(*AlarmCtrl*)
(*============================*)
//AlarmCtrl();
Alarm_IO();
Alarm_Others();
MisshookSensorCtrl();
(*Arm2MisshookSensorCtrl();*)
DeactivateCtrl();

(*AnalogCtrl*)
(*============================*)
(*BrensonGen_AnalogDigitalCtrl();*)
(*BrensonMultiFreq_Main();*)
(*USFeedbackCtrl();*)
ClangsonicUSCommCtrl();
ClangsonicUSCtrl();
ModbusControl_ST();
MegasonicModbusProgram_ST();
ClangsonicUSModbusFeedbackCtrl();
ConductivityCtrl();
FilterPressureCtrl();
TempChillerCtrl();
TempCtrl();
PID_TempCtrl();
//PIDCtrl();

(*AutoArmCtrl*)
(*============================*)
VertCoERead();
HorzCoeRead();
SlowpullCoeRead();
OmronServoEnable();
AxisHorzAdditionalInterlock_Arm1();
AxisServoCtrl_SlowPull();
oArmSlowPullHomingCtrl();
oArmSlowPullOutputCtrl();
PosConfirmBitCtrl_SlowPull();

AxisHorzMovementOutputCtrl_Arm1();
AxisServoCtrl_Arm1();
AxisServoCtrlMapping_Arm1();
AxisVertMovementOutputCtrl_Arm1();
PnpCtrl_Arm1();
PnpMapping_Arm1();
PnPstorageMemory_Arm();
PosConfirmBitCtrl_Arm1();

(*PosConfirmBitCtrl_SlowPull();*)
(*AxisHorzAdditionalInterlock_Arm1();*)
(*AxisHorzOutputCtrlInterlockingST_Arm1();*)
(*AxisMovementOutputCtrl_SlowPull();*)
(*AxisServoCtrl_SlowPull();*)
(*AutoProcessCtrl*)

(*============================*)
LdBasketMissingCtrl();
LdPrcs();
LdPrcs_General();
Stn1();
Stn2();
Stn3();
Stn4();
Stn5();
Stn6();
Stn7();
Stn7ReturnPumpCtrl();
Stn8();
Stn9();
Stn9SlowPullCalculation();
Stn10();
//Lift_N_Shuttle();
BarcodeCtrl_Utac();
BarcodeScanner();
Cascading();
StnOverflowValveCtrl();

(*AutoSevenDayOnOffCtrl*)
(*============================*)
SevenDayCtrl();
SevenDayOnOffConf();

(*BaseWork*)
(*============================*)
TowerLightCtrl();
UserCtrl();

(*BasketMemory_RecipeCtrl*)
(*============================*)
BasketBadCtrl();
BasketMemoryCtrl();
BasketToleranceCtrl();
BskMemoryCtrl();
CvMotorREFE();

(*BlowerCtrl*)
(*============================*)
//BlowerCtrl();

(*DataManagement*)
(*============================*)
ArmPickTransferCtrl_General();
BasketTotalizer();
MacOperationTimeCtrl();
RTClockCtrl();
StnBasketTotalizer();

(* CSV *)
Batch_Number_counter();
Csv_Report_Ctrl();
Csv_Report_Mapping();

(*DataManagement_Barcode*)
(*============================*)
//Batch_Number_counter();
//GeneratorComparison();
Log_BasketTimeInOut();
Log_Configuration();
Log_Management();

(*DosingPumpCtrl*)
(*============================*)
ManualDosingSTreset();
Stn1DosingPumpCtrl();
(*Stn2DosingPumpCtrl();*)
Stn3DosingPumpCtrl();
(*Stn4DosingPumpCtrl();*)
Stn5DosingPumpCtrl();

(*ManualCtrl*)
(*============================*)
ManualButtonCtrl();
ManualCtrl();
ManualCtrl_Arm();
ManualLifterJog();

(*Other*)
(*============================*)
ArmXYPosAdjust();
BeckhoffHMIMapping();
HMI_Function();
HoldingBit_DoorTransfer();
HoldingBitCtrl();
(*IndusoftBeckhoffMapping();*)
ProHMIMapping();
TactTime();
zHMIMaxMinLimit();
ClockPulse10ms();

(*OutputCtrl*)
(*============================*)
MAIN_Arm_Mapping();
MP_1_Y100();
MP_2_Y101();
MP_3_Y102();
MP_4_Y103();
SP1_1_Y110();
SP1_2_Y111();
SP2_1_Y120();
SP3_1_Y130();
SP3_2_Y131();
SP3_3_Y132();
STN_TopUpCtrl();


(*TimeOptimize*)
(*============================*)
Optimizer_Monitor();
TimeOptimizeCtrl();
TimeTrackerCtrl();

(*HMI*)
HMI_Ctrl();
StartStop();

HMI_CKK();


(*xml_Function*)
(*============================*)
//Xml_AddressMapping();
//XML_Program();
pouXMLRecipeTest();




	tPowerOnDelayOn(IN:=TRUE , PT:=T#5S , Q=> , ET=> );
	tPowerOnDelayOff(IN:=tPowerOnDelayOn.Q , PT:=t#2s , Q=> , ET=> );
	
	IF bRecipeLoadPB OR (tPowerOnDelayOn.Q AND NOT tPowerOnDelayOff.Q) THEN
	bRecipeLoadInternal := TRUE;
	bRecipeLoadPB := FALSE;
	ELSE
	bRecipeLoadInternal := FALSE;
	END_IF

//END_IF

END_PROGRAM

// ---- POUs/MainProgram/XML/Bootup_Shutdown_ctrl.TcPOU
PROGRAM Bootup_Shutdown_ctrl
VAR
	bIpcInput_on: BOOL;
	bXmlReadEn: BOOL;
	bCSVReadEn: BOOL;
	bCsvReadDone: BOOL;
	
	bIPCInputOnRE	: R_trig;
	bIPCOnRE		: R_Trig;
	bXmlCsvReadDoneRE : R_Trig;
	bXmlCsvWriteDoneRE	:R_trig;
	
	bCsvWriteEn: BOOL;
	bIpcOnHR: BOOL;


	
	bSFQTest: BOOL;
	bSFQTest_read: BOOL;
	

	bBootUpReadXMLDone	:BOOL;
	bShutdownWriteXMLDone	:BOOL;
	sStatus: STRING;
	bsyed: BOOL;
	bIpcOffDelay: BOOL;
	tIpcOffDelay: TON;
	test: Bool;
	
	
	
	
	
	
	
	

	
	
	
	
	bSHutdownTest: BOOL;
	
	on: BOOL;


END_VAR

VAR PERSISTENT
	bBootupHold: BOOL;
END_VAR


// IPC OFF Selector Switch - OFF
bIPCInputOnRE(CLK:=ARbDI[eX11111_IpcDcOnSignal] OR bBatteryModeActivated OR bSFQTest , Q=> );

IF ARbDI[eX11111_IpcDcOnSignal] THEN
	on:= FALSE;
	ELSE
	on:= TRUE;
	
END_IF


// IPC autoboot start signal
bIPCOnRE(CLK:=TRUE OR bSFQTest_read  , Q=> );

//IPC On Holding relay -output
IF PowerOnDelay.Q AND NOT tIpcOffDelay.Q THEN
	bIpcOnHR := TRUE;
	ELSE
	bIpcOnHR := FALSE;
END_IF

ARwDO[eY11007_IpcDcOnHoldingRelay].00:=bIpcOnHR OR bsyed;

// Bootup
IF bIPCOnRE.Q AND NOT bBootupHold THEN
	bMainCtrl:=FALSE;
	bReadXmlEn:= TRUE;
END_IF

bXmlCsvReadDoneRE(CLK:= bReadXmlComplete (*AND NOT Alarm_XMLReadnWrite.fbXmlSrvReadFromXML.bBusy AND bCsvReadDone*) , Q=> );

IF bXmlCsvReadDoneRE.Q THEN 
	bMainCtrl:=TRUE;
	bBootupHold:= TRUE;
END_IF

// Shutdown
IF bIPCInputOnRE.Q OR bSHutdownTest THEN
	bBootupHold:= FALSE;
	bMachineShutdown:=TRUE;
	bShutdownPopupPage:=TRUE;
	bRecipeShutdownRequestFlag:= TRUE;
	bCsvShutdownRequestFlag:=TRUE;
	bWriteXmlEn:= TRUE;
END_IF

bXmlCsvWriteDoneRE(CLK:= bWrite_Done (*AND bRecipeReadyToShutdownFlag AND bCsvReadyToShutdownFlag*), Q=> );

IF bXmlCsvWriteDoneRE.Q THEN
	bIpcOffDelay:= TRUE;
	bWriteXmlEn:=FALSE;
	
END_IF

tIpcOffDelay(IN:=bIpcOffDelay , PT:= T#2S , Q=> , ET=> );

END_PROGRAM

// ---- POUs/MainProgram/Barcode/SerialCom.TcPOU
PROGRAM SerialCom
VAR
	fbSerialControl : SerialLineControlADS;
	fbSendString	: SendString;
	fbReceiveString	: ReceiveString;
	
	bBarcodeReceivedReset_FE: F_TRIG;
END_VAR

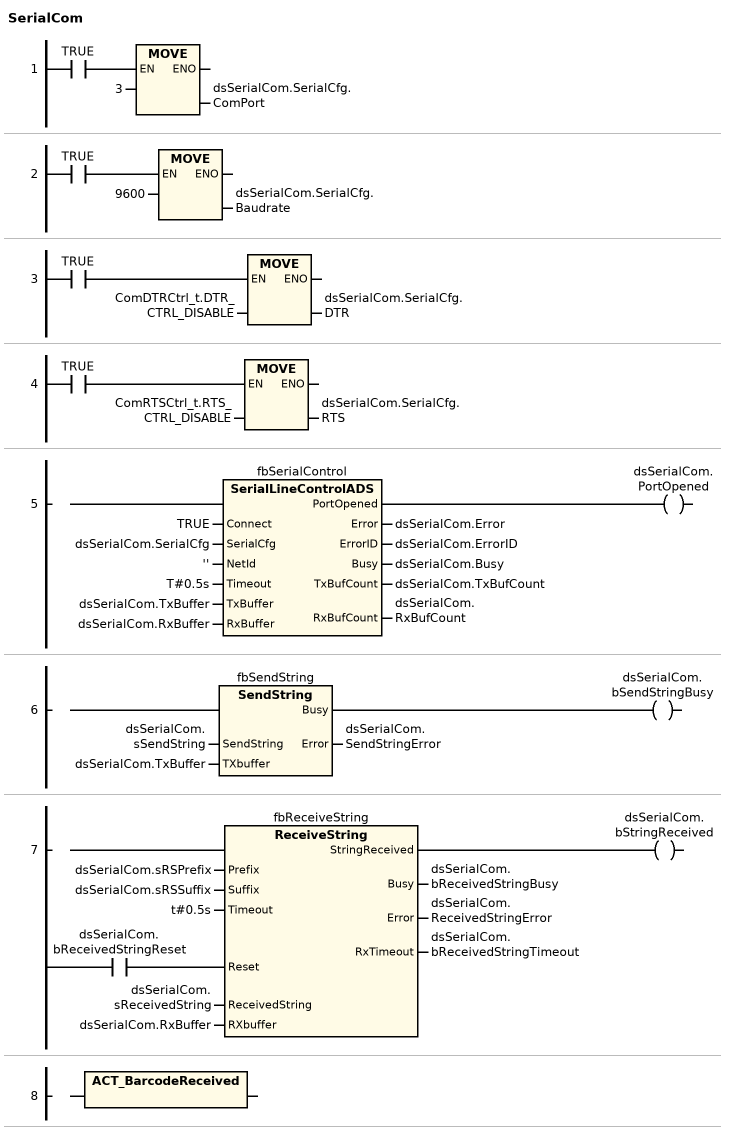
// NETWORK 1
dsSerialCom.SerialCfg.ComPort := 3;

// NETWORK 2
dsSerialCom.SerialCfg.Baudrate := 9600;

// NETWORK 3
dsSerialCom.SerialCfg.DTR := ComDTRCtrl_t.DTR_CTRL_DISABLE;

// NETWORK 4
dsSerialCom.SerialCfg.RTS := ComRTSCtrl_t.RTS_CTRL_DISABLE;

// NETWORK 5
fbSerialControl(
    Connect := TRUE,
    SerialCfg := dsSerialCom.SerialCfg,
    NetId := '',
    Timeout := T#0.5s,
    TxBuffer := dsSerialCom.TxBuffer,
    RxBuffer := dsSerialCom.RxBuffer,
    Error => dsSerialCom.Error,
    ErrorID => dsSerialCom.ErrorID,
    Busy => dsSerialCom.Busy,
    TxBufCount => dsSerialCom.TxBufCount,
    RxBufCount => dsSerialCom.RxBufCount); // SerialLineControlADS
dsSerialCom.PortOpened := fbSerialControl.PortOpened;

// NETWORK 6
fbSendString(
    SendString := dsSerialCom.sSendString,
    TXbuffer := dsSerialCom.TxBuffer,
    Error => dsSerialCom.SendStringError); // SendString
dsSerialCom.bSendStringBusy := fbSendString.Busy;

// NETWORK 7
fbReceiveString(
    Prefix := dsSerialCom.sRSPrefix,
    Suffix := dsSerialCom.sRSSuffix,
    Timeout := t#0.5s,
    Reset := dsSerialCom.bReceivedStringReset,
    ReceivedString := dsSerialCom.sReceivedString,
    RXbuffer := dsSerialCom.RxBuffer,
    Busy => dsSerialCom.bReceivedStringBusy,
    Error => dsSerialCom.ReceivedStringError,
    RxTimeout => dsSerialCom.bReceivedStringTimeout); // ReceiveString
dsSerialCom.bStringReceived := fbReceiveString.StringReceived;

// NETWORK 8
ACT_BarcodeReceived();

ACTION ACT_BarcodeReceived:

bBarcodeReceivedReset_FE(CLK:=((bAutoStartPb AND ARbDI[eX14000_LoadingConveyorSensor_Feed]) OR bBarcodeRegPage), Q=> );

IF bBarcodeReceivedReset_FE.Q THEN
dsSerialCom.sReceivedString:='';
END_IF
END_ACTION

END_PROGRAM

// ---- POUs/MainProgram/OPC_UA/OPC_UA_MAP.TcPOU
PROGRAM OPC_UA_MAP
VAR
	bIPC_Machine_Run: BOOL;
	bIPC_Machine_Alarm: BOOL;
	bIPC_Ideal_Cycle_Time: INT;


END_VAR

bMachine_Run_OPC_UA 	:=bAutoStartPb;			
                                    
                                    
bMachine_Idle_OPC_UA 	:=ARwDO[eY11005_GeneralTowerLightInd_Yellow].00;			
                                    
                                    
bMachine_Alarm_OPC_UA 	:=ARwDO[eY11004_GeneralTowerLightInd_Red].00;			
                                    
                                    
iRecipe_Number_OPC_UA 	:=iUserDefineProductRecipeNo;				
                                    
                                    
sUsername_OPCUA 		:=fbHmiTF1800_UserlevelManagement.dsHmiUserStatus_Active.sLoginName;				
                                    
                                    
ARbBasketAvailibility_OPCUA[1]:= DSStnBasketInfo[1].bAvailibility;			
ARbBasketAvailibility_OPCUA[2]:= DSStnBasketInfo[2].bAvailibility;;
ARbBasketAvailibility_OPCUA[3]:= DSStnBasketInfo[3].bAvailibility;;
ARbBasketAvailibility_OPCUA[4]:= DSStnBasketInfo[4].bAvailibility;;
ARbBasketAvailibility_OPCUA[5]:= DSStnBasketInfo[5].bAvailibility;;
ARbBasketAvailibility_OPCUA[6]:= DSStnBasketInfo[6].bAvailibility;;
ARbBasketAvailibility_OPCUA[7]:= DSStnBasketInfo[7].bAvailibility;;
ARbBasketAvailibility_OPCUA[8]:= DSStnBasketInfo[8].bAvailibility;;
ARbBasketAvailibility_OPCUA[9]:= DSStnBasketInfo[9].bAvailibility;;
//ARbBasketAvailibility_OPCUA[10]:= DSStnBasketInfo[10].bAvailibility;;
                                    
                                    
ARbStationBasketStatus_OPCUA[1]:=DSStnBasketInfo[1].sProductQuality;			
ARbStationBasketStatus_OPCUA[2]:=DSStnBasketInfo[2].sProductQuality;                                    
ARbStationBasketStatus_OPCUA[3]:=DSStnBasketInfo[3].sProductQuality;                                    
ARbStationBasketStatus_OPCUA[4]:=DSStnBasketInfo[4].sProductQuality;
ARbStationBasketStatus_OPCUA[5]:=DSStnBasketInfo[5].sProductQuality;
ARbStationBasketStatus_OPCUA[6]:=DSStnBasketInfo[6].sProductQuality;
ARbStationBasketStatus_OPCUA[7]:=DSStnBasketInfo[7].sProductQuality;
ARbStationBasketStatus_OPCUA[8]:=DSStnBasketInfo[8].sProductQuality;
ARbStationBasketStatus_OPCUA[9]:=DSStnBasketInfo[9].sProductQuality;
//ARbStationBasketStatus_OPCUA[10]:=DSStnBasketInfo[10].sProductQuality;

                                    
                                    
ARrStnTempPV_OPCUA					:=ARrStnTempPV;                                
                                  
ARrStnTempHysterysisSV_OPCUA		:=ARrStnTempHYSsv;			                                    	
                                    
ARrStnTempHighTempSV_OPCUA			:=ARrStnTempHALsv;			                                  	
                                    
ARrStnTempSV_OPCUA					:=ARrStnTempSV;					                                    
                                    
ARrStnTempReadySV_OPCUA				:=ARrStnTempRDYsv;		                                    
                                    
ARrStnTemp1stLimitSV_OPCUA			:=ARrStnTemp1stLimitSv;	
                                   
ARrStnTemp2ndLimitSV_OPCUA			:=ARrStnTemp2ndLimitSv;		                                    
                                 
ARiStnPreparationTempSV_OPCUA		:=ARiStnPreparationTempSv;
                                                                      
ARrStnConductivityPV_OPCUA 			:=ARrStnConductivityPV;
                                                                      
ARrStnLowConductivitySV_OPCUA		:=ARrStnLowConductivitySv;	                                    
                                    
ARrStnHighConductivitySV_OPCUA		:=ARrStnHighConductivitySv;
                                   
ARrStnFilterPressurePV_OPCUA		:=ARrStnFilterPressurePV;
                                   
ARrStnLowFilterPressureSV_OPCUA		:=ARrStnLowFilterPressureSv;
                                   
                                   
ARrStnHighFilterPressureSV_OPCUA	:=ARrStnHighFilterPressureSv;
                                    
                                    
ARiUltrasonicPV_OPCUA[1]			:=ARiUsPowerPV_percent[1];					
ARiUltrasonicPV_OPCUA[2]			:=ARiUsPowerPV_percent[2];	
ARiUltrasonicPV_OPCUA[3]			:=ARiUsPowerPV_percent[3];	
ARiUltrasonicPV_OPCUA[4]			:=ARiUsPowerPV_percent[4];	
ARiUltrasonicPV_OPCUA[5]			:=ARiUsPowerPV_percent[5];	
ARiUltrasonicPV_OPCUA[6]			:=ARiUsPowerPV_percent[6];	
ARiUltrasonicPV_OPCUA[7]			:=ARiUsPowerPV_percent[7];	
ARiUltrasonicPV_OPCUA[8]			:=ARiUsPowerPV_percent[8];	
                                
                                    
ARiUltrasonicSV_OPCUA[1]			:=ARDsStnSeqProcessCtrl[1].Out_DSStnSeqProOutput.i3ProTankBtmUsAPwrPercent;					
ARiUltrasonicSV_OPCUA[2]			:=ARDsStnSeqProcessCtrl[2].Out_DSStnSeqProOutput.i3ProTankBtmUsAPwrPercent;	
ARiUltrasonicSV_OPCUA[3]			:=ARDsStnSeqProcessCtrl[3].Out_DSStnSeqProOutput.i3ProTankBtmUsAPwrPercent;	
ARiUltrasonicSV_OPCUA[4]			:=ARDsStnSeqProcessCtrl[4].Out_DSStnSeqProOutput.i3ProTankBtmUsAPwrPercent;	
ARiUltrasonicSV_OPCUA[5]			:=ARDsStnSeqProcessCtrl[5].Out_DSStnSeqProOutput.i3ProTankBtmUsAPwrPercent;	
ARiUltrasonicSV_OPCUA[6]			:=ARDsStnSeqProcessCtrl[6].Out_DSStnSeqProOutput.i3ProTankBtmUsAPwrPercent;	
ARiUltrasonicSV_OPCUA[7]			:=ARDsStnSeqProcessCtrl[7].Out_DSStnSeqProOutput.i3ProTankBtmUsAPwrPercent;
ARiUltrasonicSV_OPCUA[8]			:=ARDsStnSeqProcessCtrl[8].Out_DSStnSeqProOutput.i3ProTankBtmUsAPwrPercent;

END_PROGRAM

// ---- POUs/MainProgram/AnalogCtrl/Modbus_test.TcPOU
PROGRAM Modbus_test
VAR
	wReadWord :WORD;
	wWriteWord :WORD;
	
	ReadUnitID :BYTE;
	ReadModbussRegisterAdrress : INT;
	WriteModbussRegisterAdrress : INT;	
	bStart: BOOL;
	iClangStepDelaySVns : INT;
	iTimeout_Sec : INT;

	DSClangsonicGenerator : DSV2_ClangsonicGenerator;


	bModbusReadBusy: BOOL;
	bModbusWriteBusy: BOOL;
	bModbusReadError: BOOL;
	bModbusWriteError: BOOL;
	ErrorId_Read: MODBUS_ERRORS;
	ErrorId_Write: MODBUS_ERRORS;
	iStep: INT;
	iAddCounter: INT;


	ClangsonicModbus:ModbusRtuMaster_KL6x22B;
	bModbusWriteSt: BOOL;
	bModbusReadSt: BOOL;
END_VAR

ClangsonicModbus.ReadRegs(
	UnitID			:= ReadUnitID,
	Quantity		:= 1,
	MBAddr			:= INT_TO_WORD(ReadModbussRegisterAdrress),
	cbLength		:= SIZEOF	(wReadWord),
	pMemoryAddr		:= ADR		(wReadWord),
	Execute			:= bModbusReadSt,
	Timeout			:= INT_TO_TIME(iTimeout_Sec*1000),
	BUSY			=> bModbusReadBusy,
	Error			=> bModbusReadError,
	ErrorId			=> ErrorId_Read ,
	cbRead			=> );

ClangsonicModbus.WriteSingleRegister(
	UnitID			:= ReadUnitID,
	Quantity		:= 1,
	MBAddr			:= 	INT_TO_WORD(WriteModbussRegisterAdrress),
	cbLength		:= SIZEOF	(wWriteWord),
	pMemoryAddr		:= ADR		(wWriteWord),
	Execute			:= bModbusWriteSt,
	Timeout			:= INT_TO_TIME(iTimeout_Sec*1000),
	BUSY			=> bModbusWriteBusy,
	Error			=> bModbusWriteError,
	ErrorId			=> ErrorId_Write ,
	cbRead			=> );

END_PROGRAM

// ---- POUs/MainProgram/Barcode/Barcode_Reg.TcPOU
PROGRAM Barcode_Reg
VAR
	bBarcodeRegSaveRE: R_TRIG;
	iBarcodeRegUserSelectNoDataToSave_Previous: INT;
	iFL: INT;
	bBarcodeRegClearRE: R_TRIG;
	bBarcodeRegSaveTimer: TON;
	bBarcodeRegClearTimer: TON;
	bBarcodeRegSaveHR: BOOL;
	bBarcodeRegClearHR: BOOL;
	bBarcodeRegSelectEn: BOOL;
	iScanFL	: INT;
	bBarcodeDuplicate : BOOL;
	sStatus	: STRING;
	iDonNow: INT;
	sBarcodeScannerReceivedCmdForRegBuffer: STRING;
	bReceivedNewBarcodeReg: BOOL;
	bBarcodeReceived_RE: R_TRIG;
END_VAR

(*xxxxxxxxxxxxxxxxxxxxxxxxxxxxxxxxxxxxxxxxxxxxxxxxxxxxxxxxxxxxxxxxxxxxxxxxxx*)
// Check barcode duplicate
bBarcodeDuplicate := FALSE;
IF sBarcodeScannerReceivedCmdForReg <> '' THEN
		iScanFL := 1;
		FOR iScanFL := 1 TO iBarcodeRegQty DO
			IF iScanFL >= 1 AND iScanFL <= iBarcodeRegQty THEN
				IF iScanFL <> iBarcodeRegUserSelectNoDataToSave THEN 
					 IF	DsAr1sG_BarcodeRegistration[iScanFL].sBarcodeRegistered = sBarcodeScannerReceivedCmdForReg THEN
//					IF DsAr1sG_BarcodeRegSectionDisplayHMI[iScanFL].sBarcodeRegistered = sBarcodeScannerReceivedCmdForReg THEN
						bBarcodeDuplicate := TRUE;
						iDonNow:=iScanFL;
					END_IF
				END_IF
			END_IF
		END_FOR
END_IF

// Error Status shown when Barcode detected was ERROR
IF bBarcodeDuplicate THEN
iScanFL := 1;
FOR iScanFL := 1 TO iBarcodeRegQty DO
	IF iScanFL >= 1 AND iScanFL <= iBarcodeRegSecDisplayQty THEN
		sStatus := 'Error - Barcode Duplicated Found. Make sure assign barcode correctly';
		iScanFL := iBarcodeRegQty+1;
	END_IF
END_FOR
ELSE
		sStatus := 'No Error Found';
END_IF

// Barcode scanner received push to buffer barcode for register
IF sBarcodeScannerReceivedCmd <> '' AND sBarcodeScannerReceivedCmdForRegBuffer<>sBarcodeScannerReceivedCmd AND bBarcodeRegPage  THEN
sBarcodeScannerReceivedCmdForRegBuffer := sBarcodeScannerReceivedCmd;
bReceivedNewBarcodeReg:=TRUE;
ELSE
bReceivedNewBarcodeReg:=FALSE;
END_IF

bBarcodeReceived_RE(CLK:=bReceivedNewBarcodeReg , Q=> );
	
IF bBarcodeReceived_RE.Q THEN
	sBarcodeScannerReceivedCmdForReg:=sBarcodeScannerReceivedCmdForRegBuffer;
END_IF

IF NOT bBarcodeRegPage THEN
	sBarcodeScannerReceivedCmdForReg:='';
	sBarcodeScannerReceivedCmdForRegBuffer:='';
END_IF

IF sBarcodeScannerReceivedCmdForReg = '' THEN
bBarcodeEmpty := TRUE;
ELSE
bBarcodeEmpty := FALSE;
END_IF

// Barcode reg control
bBarcodeRegSaveRE(CLK:=bBarcodeRegSave , Q=> );
bBarcodeRegClearRE(CLK:=bBarcodeRegClear , Q=> );
bBarcodeRegSaveTimer(IN:=bBarcodeRegSaveHR , PT:=T#0.5S , Q=> , ET=> );
bBarcodeRegClearTimer(IN:=bBarcodeRegClearHR , PT:=T#0.5S , Q=> , ET=> );

IF bBarcodeRegSaveTimer.Q THEN
	bBarcodeRegSaveHR := FALSE;
END_IF

IF bBarcodeRegClearTimer.Q THEN
	bBarcodeRegClearHR := FALSE;
END_IF

IF bBarcodeRegSaveRE.Q THEN
	bBarcodeRegSaveHR := TRUE;
END_IF

IF bBarcodeRegClearRE.Q THEN
	bBarcodeRegClearHR := TRUE; 
END_IF

IF bBarcodeRegSaveHR OR bBarcodeRegClearHR 
OR iBarcodeRegUserSelectNoDataToSave_Previous <> iBarcodeRegUserSelectNoDataToSave 
THEN
bBarcodeReceiveStringRst			:= TRUE ;
ELSE
bBarcodeReceiveStringRst			:= FALSE ;
END_IF


bBarcodeRegSelectEn := iBarcodeRegUserSelectNoDataToSave <> 0;

		IF bBarcodeRegSaveRE.Q AND NOT bBarcodeDuplicate AND sBarcodeScannerReceivedCmdForReg <> '' AND iBarcodeRegUserSelectRecipeNo <> 0 THEN
	 		IF iBarcodeRegUserSelectNoDataToSave >= 1 AND iBarcodeRegUserSelectNoDataToSave <= iBarcodeRegQty THEN
				DsAr1sG_BarcodeRegistration[iBarcodeRegUserSelectNoDataToSave].iLinkProductRecipeNo				:= iBarcodeRegUserSelectRecipeNo;
				//DsAr1sG_BarcodeRegistration[iBarcodeRegUserSelectNoDataToSave].sLinkProductRecipeNoDisplay		:= TO_STRING(iBarcodeRegUserSelectRecipeNo);
				DsAr1sG_BarcodeRegistration[iBarcodeRegUserSelectNoDataToSave].sBarcodeRegistered				:= sBarcodeScannerReceivedCmdForReg;
				DsAr1sG_BarcodeRegistration[iBarcodeRegUserSelectNoDataToSave].sLinkProductRecipeDescription	:= ARsProductRecipeDescription[iBarcodeRegUserSelectRecipeNo];
			END_IF
		END_IF
		IF bBarcodeRegSaveHR THEN
		iBarcodeRegUserSelectRecipeNo		:= 0	;
		sBarcodeScannerReceivedCmdForReg	:= ''	;
		iBarcodeRegUserSelectNoDataToSave 	:= 0	;		
		END_IF

		IF bBarcodeRegClearRE.Q THEN
	 		IF iBarcodeRegUserSelectNoDataToSave >= 1 AND iBarcodeRegUserSelectNoDataToSave <= iBarcodeRegQty THEN
				DsAr1sG_BarcodeRegistration[iBarcodeRegUserSelectNoDataToSave].iLinkProductRecipeNo				:=	0;
				//DsAr1sG_BarcodeRegistration[iBarcodeRegUserSelectNoDataToSave].sLinkProductRecipeNoDisplay		:=	'';
				DsAr1sG_BarcodeRegistration[iBarcodeRegUserSelectNoDataToSave].sBarcodeRegistered				:=	'';
				DsAr1sG_BarcodeRegistration[iBarcodeRegUserSelectNoDataToSave].sLinkProductRecipeDescription	:=	'';
			END_IF
		END_IF
		IF bBarcodeRegClearHR THEN
		iBarcodeRegUserSelectRecipeNo		:= 0	;
		sBarcodeScannerReceivedCmdForReg	:= ''	;
		iBarcodeRegUserSelectNoDataToSave 	:= 0	;		
		END_IF

	(*
		IF iBarcodeRegUserSelectNoDataToSave_Previous <> iBarcodeRegUserSelectNoDataToSave THEN
			iBarcodeRegUserSelectNoDataToSave_Previous := iBarcodeRegUserSelectNoDataToSave;
			FOR iFL := 1 TO iBarcodeRegQty DO
				DsAr1sG_BarcodeRegistration[iFL].bHmiBarcodeRegistrationSelected := FALSE;
			END_FOR

	 		IF iBarcodeRegUserSelectNoDataToSave >= 1 AND iBarcodeRegUserSelectNoDataToSave <= iBarcodeRegQty THEN
			
				DsAr1sG_BarcodeRegistration[iBarcodeRegUserSelectNoDataToSave].bHmiBarcodeRegistrationSelected := TRUE;
				
				iBarcodeRegUserSelectRecipeNo	:= DsAr1sG_BarcodeRegistration[iBarcodeRegUserSelectNoDataToSave].iLinkProductRecipeNo	;
				sBarcodeScannerReceivedCmdForReg:=	DsAr1sG_BarcodeRegistration[iBarcodeRegUserSelectNoDataToSave].sBarcodeRegistered	;
			END_IF			
		END_IF
		*)

END_PROGRAM

// ---- POUs/MainProgram/Mapping/Internal_Mapping.TcPOU
PROGRAM Internal_Mapping
VAR
	CKKALARMRESET: BOOL;
	CKKBUZZERRESET: BOOL;
	
END_VAR

//ARwDO[eY11002_GeneralBuzzerTone01].00:=bBuzzerOutput; // Need to mapping with pyshical Output Buzzer Tone 1

//bEventRstPBPhysicalInput:=ARbDI[eX10000_Stn01UltrasonicGeneratorMcb_Trip] OR CKKALARMRESET OR bHMI_AlarmRstPB;  // Need to mapping with physical Input Alarm Reset PB
//bBuzzerRstPBPhysicalInput:=ARbDI[eX10001_GeneralBuzzerPb_Reset] OR CKKBUZZERRESET OR bHMI_BuzzerRstPB; // Need to mapping with physical Input Buzzer Reset PB


// Clangsonic Ultrasonic Mapping
//ARdsClangsonicGenerator[1].iGenModbusUnitID		:= 1;
//ARdsClangsonicGenerator[2].iGenModbusUnitID		:= 2;
//ARdsClangsonicGenerator[3].iGenModbusUnitID		:= 3;

//ARdsClangsonicGenerator[1].iModbusRS485ChannelID	:= 1;
//ARdsClangsonicGenerator[2].iModbusRS485ChannelID	:= 1;
//ARdsClangsonicGenerator[3].iModbusRS485ChannelID	:= 1;


// Misshook Sensor

	ARbMAP_ArmMisshookSensorA[1]	:= ARbDI[eX11004_Arm01SensorA_Misshook];
	ARbMAP_ArmMisshookSensorB[1]	:= ARbDI[eX11005_Arm01SensorB_Misshook];
	

//  Last index basket at loading ( Basket LD arm pick )

	bMAP_LdConfirmBasketPickAvailibility   := AR2sDSCv_LdConfirmBasketInfo[1,3].bAvailibility;

END_PROGRAM

// ---- POUs/MainProgram/Mapping/IO_Mapping.TcPOU
PROGRAM IO_Mapping
VAR
END_VAR


//Input
 
ARwMapDI[100]:= ARwActualMapDI[1] ;
ARwMapDI[101]:= ARwActualMapDI[2] ;
ARwMapDI[102]:= ARwActualMapDI[3] ;
ARwMapDI[103]:= ARwActualMapDI[4] ;
ARwMapDI[104]:= ARwActualMapDI[5] ;
ARwMapDI[110]:= ARwActualMapDI[6] ;
ARwMapDI[111]:= ARwActualMapDI[7] ;
ARwMapDI[120]:= ARwActualMapDI[8] ;
ARwMapDI[121]:= ARwActualMapDI[9] ;
ARwMapDI[130]:= ARwActualMapDI[10];
ARwMapDI[140]:= ARwActualMapDI[11];
ARwMapDI[150]:= ARwActualMapDI[12];


FN_DigitalInputMapping(TRUE,100,1);
FN_DigitalInputMapping(TRUE,101,17);
FN_DigitalInputMapping(TRUE,102,33);
FN_DigitalInputMapping(TRUE,103,49);
FN_DigitalInputMapping(TRUE,104,65);
FN_DigitalInputMapping(TRUE,110,81);
FN_DigitalInputMapping(TRUE,111,97);
FN_DigitalInputMapping(TRUE,120,113);
FN_DigitalInputMapping(TRUE,121,129);
FN_DigitalInputMapping(TRUE,130,145);
FN_DigitalInputMapping(TRUE,140,161);
FN_DigitalInputMapping(TRUE,150,177);


//Output

FN_DigitalOutputMapping(TRUE,100,1);
FN_DigitalOutputMapping(TRUE,101,17);
FN_DigitalOutputMapping(TRUE,102,33);
FN_DigitalOutputMapping(TRUE,103,49);
FN_DigitalOutputMapping(TRUE,110,65);
FN_DigitalOutputMapping(TRUE,111,81);
FN_DigitalOutputMapping(TRUE,120,97);
FN_DigitalOutputMapping(TRUE,130,113);
FN_DigitalOutputMapping(TRUE,131,129);
FN_DigitalOutputMapping(TRUE,132,145);

ARwActualMapDO[1]:= ARwMapDO[100] ;
ARwActualMapDO[2]:= ARwMapDO[101] ;
ARwActualMapDO[3]:= ARwMapDO[102] ;
ARwActualMapDO[4]:= ARwMapDO[103] ;
ARwActualMapDO[5]:= ARwMapDO[110] ;
ARwActualMapDO[6]:= ARwMapDO[111] ;
ARwActualMapDO[7]:= ARwMapDO[120] ;
ARwActualMapDO[8]:= ARwMapDO[130] ;
ARwActualMapDO[9]:= ARwMapDO[131] ;
ARwActualMapDO[10]:= ARwMapDO[132] ;

END_PROGRAM

// ---- POUs/MainProgram/zAutoMode/AutoMain_AddON.TcPOU
PROGRAM AutoMain_AddON
VAR

	MainOnOffStartRE			:R_TRIG;
	PreparationStartRE		:R_TRIG;
	OriginStartRE				:R_TRIG;
	AutoModeRE				:R_TRIG;

	MainOnOffDelayOffTON	: TON;
	PreparationStartTON		: TON;
	OriginStartTON			:TON;
	AutoModeTON			:TON;

	bTest1	:BOOL;

END_VAR

(*To start the Main On OFF Bit*)
MainOnOffStartRE(CLK:= bMainOnOffBuff, Q=> );
IF MainOnOffStartRE.Q THEN
	bMainOnOff :=TRUE;
	bTest1:=TRUE;
END_IF

(*To Reset Main On Off bit*)
MainOnOffDelayOffTON(IN:=(bMainonOff OR bTest1) AND  bMainOnOffBuff, PT:=t#5s , Q=> , ET=> );
IF MainOnOffDelayOffTON.Q THEN
	bMainOnOff:=FALSE;
	bTest1:=FALSE;
END_IF



(*To start the Auto Preparation PB  Bit*)
PreparationStartRE(CLK:= bAutoPreparationPbBuff, Q=> );
IF PreparationStartRE.Q THEN
	bAutoPreparationPb  :=TRUE;
END_IF

(*To Reset Auto Preparation PB bit*)
PreparationStartTON(IN:= bAutoPreparationPb AND  bAutoPreparationPbBuff, PT:=t#5s , Q=> , ET=> );
IF PreparationStartTON.Q THEN
	bAutoPreparationPb:=FALSE;
END_IF




(*To start the Auto Origin PB  Bit*)
OriginStartRE(CLK:= bAutoOriginPbBuff, Q=> );
IF OriginStartRE.Q THEN
	bAutoOriginPb  :=TRUE;
END_IF

(*To Reset Auto Origin PB bit*)
OriginStartTON(IN:= bAutoOriginPbBuff AND  bAutoOriginPB, PT:=t#5s , Q=> , ET=> );
IF OriginStartTON.Q THEN
	bAutoOriginPB:=FALSE;
END_IF




(*To start the bAutoStartPb Bit*)
AutoModeRE(CLK:= bAutoStartPbBuff, Q=> );
IF AutoModeRE.Q THEN
	bAutoStartPb  :=TRUE;
END_IF

(*To Reset bAutoStartPb bit*)
AutoModeTON(IN:= bAutoStartPbBuff AND  bAutoStartPb, PT:=t#5s , Q=> , ET=> );
IF AutoModeTON.Q THEN
	bAutoStartPb:=FALSE;
END_IF


(*

	bMainOnOffBuff						:BOOL; (*Add on For Main On Off delay Off-20181112*)
	bAutoPreparationPbBuff      				: BOOL;
	bAutoOriginPbBuff						: BOOL;
	bAutoStartPbBuff						: BOOL;

	bMainOnOff							: BOOL;
	bAutoPreparationPb      				: BOOL;
	bAutoPreparationInt	      				: BOOL;
	bAutoPreparationDone					: BOOL;
	bAutoOriginPb						: BOOL;
	bAutoOriginDone						: BOOL;
	bAutoStartPb							: BOOL;

*)

END_PROGRAM

// ---- POUs/MainProgram/Other/HMI_Page_Control.TcPOU
PROGRAM HMI_Page_Control
VAR
	PowerOnDelayRE	:R_TRIG;
END_VAR

(*tLdSensor1DelayOffTimer(IN:=(NOT X120_00 ) , PT:= t#0.5s, Q=> , ET=> );*)
(*Initial Loading PAge*)
(*
bAutoModeOnTON	:TON;
	bManualModeOnTON	:TON;
	bRecipeModeOnTON	:TON;
	bRecipeSSUROnTON	:TON;
	bRecipeSSEROnTON	:TON;
	bAlarmModeOnTON	:TON;
	bUserModeOnTON	:TON;
*)
(*
bAutoModeOnTON(IN:=( NOT bAutoModeOnSeq ) , PT:= t#5s, Q=> , ET=> );
bManualModeOnTON(IN:=(bAutoModeOnSeq AND NOT bManualModeOnSeq ) , PT:= t#5s, Q=> , ET=> );
bRecipeModeOnTON(IN:=(bManualModeOnSeq AND NOT bRecipeModeOnSeq ) , PT:= t#5s, Q=> , ET=> );
bRecipeSSEROnTON(IN:=(bRecipeModeOnSeq AND NOT bRecipeSSEROnSeq ) , PT:= t#5s, Q=> , ET=> );
bRecipeSSUROnTON(IN:=(bRecipeSSEROnSeq AND NOT bRecipeSSUROnSeq ) , PT:= t#5s, Q=> , ET=> );

IF NOT bAutoModeOnTON.Q THEN
	bAutoModeOn:=TRUE;
ELSIF  bAutoModeOnTON.Q THEN
	bAutoModeOn:=FALSE;
	bAutoModeOnSeq:=TRUE;
	bManualModeOn:=TRUE;
ELSIF bManualModeOnTON.Q THEN
	bManualModeOn:=FALSE;
	bManualModeOnSeq:=TRUE;
	bRecipeModeOn:=TRUE;
	bRecipeSSEROn:=TRUE;
ELSIF bRecipeSSEROnTON.Q THEN
	bRecipeModeOn:=FALSE;
	bRecipeSSEROn:=FALSE;
	bRecipeSSEROnSeq:=TRUE;
	bRecipeSSUROn:=TRUE;
ELSIF bRecipeSSUROnTON.Q THEN
	bRecipeSSUROn:=FALSE;
	bRecipeSSUROnSeq:=TRUE;
	bLoadingPageSeqComplete:=TRUE;
END_IF

IF bLoadingPageSeqCompleteRE.Q THEN
	bAutoModeOn:=TRUE;
END_IF

*)






(*PAge Screen Changes Control*)
//Start comment - syafiq
(*PowerOnDelayRE(CLK:=  PowerOnDelay.Q, Q=> );
bAutoModeOnRE(CLK:=  bAutoModeOnPB, Q=> );
bManualModeOnRE(CLK:=  bManualModeOnPB, Q=> );

bRecipeModeOnRE(CLK:=  bRecipeModeOnPB, Q=> );
	bRecipeSSUROnRE(CLK:=  bRecipeSSUROnPB, Q=> );
	bRecipeSSEROnRE(CLK:=  bRecipeSSEROnPB, Q=> );
	bRecipeBasicOnRE(CLK:=  bRecipeBasicOnPB, Q=> );
          bRecipeBasic2OnRE(CLK:= bRecipeBasic2OnPB, Q=> );
	bRecipeProductOnRE(CLK:=  bRecipeProductOnPB, Q=> );
	bRecipeOtherOnRE(CLK:=  bRecipeOtherOnPB, Q=> );
	bRecipeTimeOptimizeOnRE(CLK:=  bRecipeTimeOptimizeOnPB, Q=> );
         bRecipeArmSettingOnRE(CLK:= bRecipeArmSettingOnPB, Q=> );
	bRecipeArmSetting2OnRE(CLK:= bRecipeArmSetting2OnPB, Q=> );

bUserModeOnRE(CLK:=  bUserModeOnPB, Q=> );
bAlarmModeOnRE(CLK:=  bAlarmModeOnPB, Q=> );
bManualModeOnLatchFE(CLK:=  bManualModeOnLatch, Q=> );

bManuPageOn:=bManualModeOnLatch;

(*Others Mode Control*)
IF NOT  bManualModeOnLatch THEN
	IF bAutoModeOnRE.Q THEN
		bAutoModeOn:=TRUE;
		bManualModeOn:=FALSE;
		bRecipeModeOn:=FALSE;
		bUserModeOn:=FALSE;
		bAlarmModeOn:=FALSE;
	ELSIF bManualModeOnRE.Q THEN
		bManualModeOn:=TRUE;
		bManualModeOnLatch:=TRUE;
		bAutoModeOn:=FALSE;
		bRecipeModeOn:=FALSE;
		bUserModeOn:=FALSE;
		bAlarmModeOn:=FALSE;
	ELSIF bRecipeModeOnRE.Q THEN
		bRecipeProductOn:=TRUE;
		bRecipeOtherOn	:=FALSE;
		bRecipeTimeOptimizeOn:=FALSE;
		bRecipeSSEROn:=FALSE;
		bRecipeSSUROn:=FALSE;
		bRecipeBasicOn:=FALSE;
                   bRecipeBasic2On:=FALSE;
                   bRecipeModeOn:=TRUE;
		bManualModeOn:=FALSE;
		bAutoModeOn:=FALSE;
		bUserModeOn:=FALSE;
		bAlarmModeOn:=FALSE;
	ELSIF bUserModeOnRE.Q THEN
		bUserModeOn:=TRUE;
		bManualModeOn:=FALSE;
		bAutoModeOn:=FALSE;
		bRecipeModeOn:=FALSE;
		bAlarmModeOn:=FALSE;
	ELSIF bAlarmModeOnRE.Q THEN
		bAlarmModeOn:=TRUE;
		bManualModeOn:=FALSE;
		bAutoModeOn:=FALSE;
		bRecipeModeOn:=FALSE;
		bUserModeOn:=FALSE;
	END_IF
END_IF


(*Recipe Mode Page Control*)
IF NOT bRecipeModeOn THEN
		bRecipeSSUROn:=FALSE;
		bRecipeSSEROn:=FALSE;
		bRecipeBasicOn:=FALSE;
                   bRecipeBasic2On:=FALSE;
                  bRecipeProductOn:=FALSE;
		bRecipeOtherOn	:=FALSE;
		bRecipeTimeOptimizeOn:=FALSE;
		bRecipeArmSettingOn:=FALSE;
		bRecipeArmSetting2On:=FALSE;
	ELSIF bRecipeModeOn AND bRecipeSSUROnRE.Q THEN
		bRecipeSSUROn:=TRUE;(*ON*)
		bRecipeSSEROn:=FALSE;
		bRecipeBasicOn:=FALSE;
                  bRecipeBasic2On:=FALSE;
                   bRecipeProductOn:=FALSE;
		bRecipeOtherOn	:=FALSE;
		bRecipeTimeOptimizeOn:=FALSE;
		bRecipeArmSettingOn:=FALSE;
		bRecipeArmSetting2On:=FALSE;
	ELSIF bRecipeModeOn AND bRecipeSSEROnRE.Q THEN
		bRecipeSSEROn:=TRUE;(*ON*)
		bRecipeSSUROn:=FALSE;
		bRecipeBasicOn:=FALSE;
                  bRecipeBasic2On:=FALSE;
                   bRecipeProductOn:=FALSE;
		bRecipeOtherOn	:=FALSE;
		bRecipeTimeOptimizeOn:=FALSE;
		bRecipeArmSettingOn:=FALSE;
		bRecipeArmSetting2On:=FALSE;
	ELSIF bRecipeModeOn AND bRecipeBasicOnRE.Q THEN
		bRecipeBasicOn:=TRUE;(*ON*)
                   bRecipeBasic2On :=FALSE;
                   bRecipeSSUROn :=FALSE;
		bRecipeSSEROn:=FALSE;
		bRecipeProductOn:=FALSE;
		bRecipeOtherOn	:=FALSE;
		bRecipeTimeOptimizeOn:=FALSE;
		bRecipeArmSettingOn:=FALSE;
		bRecipeArmSetting2On:=FALSE;
         ELSIF bRecipeModeOn AND bRecipeBasic2OnRE.Q THEN
                   bRecipeBasicOn:=FALSE;
                   bRecipeBasic2On:=TRUE;(*ON*)
                   bRecipeSSUROn:=FALSE;
		bRecipeSSEROn:=FALSE;
		bRecipeProductOn:=FALSE;
		bRecipeOtherOn	:=FALSE;
		bRecipeTimeOptimizeOn:=FALSE;
          ELSIF bRecipeModeOn AND bRecipeProductOnRE.Q THEN
		bRecipeBasicOn:=FALSE;
                   bRecipeBasic2On:=FALSE;
                   bRecipeSSUROn:=FALSE;
		bRecipeSSEROn:=FALSE;
		bRecipeProductOn:=TRUE;(*ON*)
		bRecipeOtherOn	:=FALSE;
		bRecipeTimeOptimizeOn:=FALSE;
		bRecipeArmSettingOn:=FALSE;
		bRecipeArmSetting2On:=FALSE;
	ELSIF bRecipeModeOn AND bRecipeOtherOnRE.Q THEN
		bRecipeBasicOn:=FALSE;
                  bRecipeBasic2On:=FALSE;
                   bRecipeSSUROn:=FALSE;
		bRecipeSSEROn:=FALSE;
		bRecipeProductOn:=FALSE;
		bRecipeOtherOn	:=TRUE;(*ON*)
		bRecipeTimeOptimizeOn:=FALSE;
		bRecipeArmSettingOn:=FALSE;
		bRecipeArmSetting2On:=FALSE;
	ELSIF bRecipeModeOn AND bRecipeTimeOptimizeOnRE.Q THEN
		bRecipeBasicOn:=FALSE;
                   bRecipeBasic2On:=FALSE;
                   bRecipeSSUROn:=FALSE;
		bRecipeSSEROn:=FALSE;
		bRecipeProductOn:=FALSE;
		bRecipeOtherOn	:=FALSE;
		bRecipeTimeOptimizeOn:=TRUE;(*ON*)
		bRecipeArmSettingOn:=FALSE;
		bRecipeArmSetting2On:=FALSE;
	ELSIF bRecipeModeOn AND bRecipeArmSettingOnRE.Q THEN
		bRecipeBasicOn:=FALSE;
                   bRecipeBasic2On:=FALSE;
                   bRecipeSSUROn:=FALSE;
		bRecipeSSEROn:=FALSE;
		bRecipeProductOn:=FALSE;
		bRecipeOtherOn	:=FALSE;
		bRecipeTimeOptimizeOn:=FALSE;
		bRecipeArmSettingOn:=TRUE;(*ON*)
		bRecipeArmSetting2On:=FALSE;
ELSIF bRecipeModeOn AND bRecipeArmSetting2OnRE.Q THEN
		bRecipeBasicOn:=FALSE;
                   bRecipeBasic2On:=FALSE;
                   bRecipeSSUROn:=FALSE;
		bRecipeSSEROn:=FALSE;
		bRecipeProductOn:=FALSE;
		bRecipeOtherOn	:=FALSE;
		bRecipeTimeOptimizeOn:=FALSE;
		bRecipeArmSettingOn:=FALSE;
		bRecipeArmSetting2On:=TRUE;(*ON*)

END_IF

(*bRecipeProductOn:BOOL;
		bRecipeOtherOn	:BOOL;
		bRecipeTimeOptimizeOn:BOOL;*)

(*Manual Mode Page Control*)
IF bManualModeOnLatch THEN
	IF bAutoModeOnRE.Q THEN
		bManualOutToAutoConfirmPageOn:=TRUE;
	ELSIF bManualModeOnLatch AND bRecipeModeOnRE.Q THEN
		bManualOutToRecipeConfirmPageOn:=TRUE;
	ELSIF bManualModeOnLatch AND bUserModeOnRE.Q THEN
		bManualOutToUserConfirmPageOn:=TRUE;
	ELSIF bManualModeOnLatchFE.Q THEN
		bAutoModeOnPB:=FALSE;
		bManualModeOnPB:=FALSE;
		bRecipeModeOnPB:=FALSE;
	ELSIF bAlarmModeOnRE.Q THEN
		bAlarmModeOn:=TRUE;
		bManualModeOn:=FALSE;
		bAutoModeOn:=FALSE;
		bRecipeModeOn:=FALSE;
		bUserModeOn:=FALSE;
	ELSIF bManualModeOnRE.Q THEN
		bManualModeOn:=TRUE;
		bManualModeOnLatch:=TRUE;
		bAutoModeOn:=FALSE;
		bRecipeModeOn:=FALSE;
		bUserModeOn:=FALSE;
		bAlarmModeOn:=FALSE;
	END_IF
ELSE bManualOutToAutoConfirmPageOn:=FALSE;
	bManualOutToRecipeConfirmPageOn:=FALSE;
	bManualOutToUserConfirmPageOn:=FALSE;
	bManualCalibrate:=FALSE;
END_IF





IF bManualModeOnLatchFE.Q THEN
	bManualOutLatchCfm:=TRUE;

END_IF

bManualOutLatchCfmTON(IN:= bManualOutLatchCfm, PT:= t#1s , Q=> , ET=> );

IF bManualOutLatchCfmTON.Q THEN
	bAutoModeOnPB:=FALSE;
	bRecipeModeOnPB:=FALSE;
	bUserModeOnPB:=FALSE;
	bManualOutLatchCfm:=FALSE;

END_IF


IF NOT bAutoModeOn THEN
	bAutoPrepareStatus:=FALSE;
	bStatusOriginPageOn:=FALSE;
	bStatusPreparePageOn:= FALSE;
	bBarcodeRegisterPageON:=FALSE;
	bSecGemsPageON:=FALSE;

END_IF

*)
// end comment - Syafiq

(*Save confirmation page ctrl*)
bSavePageCnfmOnRE(CLK:=  bSaveCfmPB, Q=> );
bSaveBufferPBRE(CLK:=  bSaveBufferPB, Q=> );

IF bSavePageCnfmOnRE.Q THEN
	bSaveCfmPageOn:=TRUE;

END_IF
(*
IF (sUserPasswordSave = UserPassword[6]) OR (sUserPasswordSave = UserPassword[7]) AND bSaveBufferPBRE.Q THEN
bRecipeSavePb:=TRUE;
bIncorrectPswdOn:=FALSE;
END_IF

IF (sUserPasswordSave <> UserPassword[6]) AND (sUserPasswordSave <> UserPassword[7]) AND bSaveBufferPBRE.Q THEN
bIncorrectPswdOn:=TRUE;
END_IF

tBackupDelayOffTimer(IN:=bRecipeSavePb, PT:=t#1s , Q=> , ET=> );

IF tBackupDelayOffTimer.Q THEN
	bRecipeSavePb:=FALSE;
END_IF
*)
IF tBackupDelayOffTimer.Q THEN
	bSaveCfmPageOn:=FALSE;
	sUserPasswordSave:='';
	bIncorrectPswdOn:=FALSE;
END_IF


(*Door Control Auto Mode*)
(*
IF bStn1DoorOpenCompleted THEN
	wDoorOpenFunc.1:=FALSE;
ELSIF  bStn1DoorCloseCompleted THEN
	wDoorCloseFunc.1:=FALSE;
END_IF


(*Door Motor Brake Release*)
IF Y100_14 OR Y100_15 THEN
	WY10204_01:=TRUE;
ELSE WY10204_01:=FALSE;
END_IF
*)

END_PROGRAM

// ---- POUs/MainProgram/A_StandardStructureProgram/stClockPulseBlink.TcPOU
PROGRAM stClockPulseBlink
VAR
	tClockPulse_1SecTimer: TON;
	bClockPulse_1SecRE: R_TRIG;

	tClockPulse_0_5SecTimer: TON;
	bClockPulse_0_5SecRE: R_TRIG;

	tClockPulse_0_1SecTimer: TON;
	bClockPulse_0_1SecRE: R_TRIG;
	
	tClockPulse_10msTimer: TON;
	bClockPulse_10msRE: R_TRIG;
	
	tClockBlink_1SecTimerA: TON;
	tClockBlink_1SecTimerB: TON;
END_VAR


// Clock Pulse - 1 Sec
tClockPulse_1SecTimer(IN:= NOT tClockPulse_1SecTimer.Q , PT:=T#1S , Q=> , ET=> );
bClockPulse_1SecRE(CLK:=tClockPulse_1SecTimer.Q , Q=> );
bClockPulse_1Sec := bClockPulse_1SecRE.Q;

// Clock Pulse - 0.5 Sec
tClockPulse_0_5SecTimer(IN:= NOT tClockPulse_0_5SecTimer.Q , PT:=T#0.5S , Q=> , ET=> );
bClockPulse_0_5SecRE(CLK:=tClockPulse_0_5SecTimer.Q , Q=> );
bClockPulse_0_5Sec := bClockPulse_0_5SecRE.Q;

// Clock Pulse - 0.1 Sec
tClockPulse_0_1SecTimer(IN:= NOT tClockPulse_0_1SecTimer.Q , PT:=T#0.1S , Q=> , ET=> );
bClockPulse_0_1SecRE(CLK:=tClockPulse_0_1SecTimer.Q , Q=> );
bClockPulse_0_1Sec := bClockPulse_0_1SecRE.Q;

// Clock Pulse - 10 ms
tClockPulse_10msTimer(IN:= NOT tClockPulse_10msTimer.Q , PT:=T#10MS , Q=> , ET=> );
bClockPulse_10msRE(CLK:=tClockPulse_10msTimer.Q , Q=> );
bClockPulse_10ms := bClockPulse_10msRE.Q;

// Clock Blink - 1 Sec (0.5Sec ON <-> 0.5Sec OFF)
tClockBlink_1SecTimerA(IN:= NOT tClockBlink_1SecTimerB.Q , PT:=T#0.5S , Q=> , ET=> );
tClockBlink_1SecTimerB(IN:= tClockBlink_1SecTimerA.Q , PT:=T#0.5S , Q=> , ET=> );
bClockBlink_1Sec := tClockBlink_1SecTimerA.Q;

END_PROGRAM

// ---- POUs/MainProgram/A_StandardStructureProgram/stGetCurrentTime.TcPOU
PROGRAM stGetCurrentTime
VAR

	LocalSystemTime			: FB_LocalSystemTime;


	sLangDayOfWeek 			: ARRAY [1..C_iLanguageQty, 0..6] OF STRING;
	sLangMonth 				: ARRAY [1..C_iLanguageQty, 1..12] OF STRING;
	sLangAmPm 				: ARRAY [1..C_iLanguageQty, 1..2] OF STRING;
                                         
	bOneScanRE				: R_TRIG;
	


	bOverrideCurrentDate: BOOL;
END_VAR

	(*---------------------------OUTPUT---------------------------------------------*)
	(*DISPLAY FORMAT - General Format*)

	DSLocalSystemTimeML.dtCurrentDateTime; 			// Newly Added *Standard DATE_AND_TIME format
	DSLocalSystemTimeML.sCurrentDateTime; 			// Newly Added *Follow standard DATE_AND_TIME format and take out " DT# "
	DSLocalSystemTimeML.sCurrentDate_General; 		// Newly Added
	DSLocalSystemTimeML.sCurrentTime24Hr_General; 	// Newly Added

	DSLocalSystemTimeML.sCurrentDT24Hr_General;

	
	(*DISPLAY FORMAT - MultiLanguage*)
	DSLocalSystemTimeML.sCurrentDT12Hr;
	DSLocalSystemTimeML.sCurrentDT24Hr;
	
	DSLocalSystemTimeML.sDayOfWeek;
	
	DSLocalSystemTimeML.sYear;
	DSLocalSystemTimeML.sMonth;
	DSLocalSystemTimeML.sDay;
	
	DSLocalSystemTimeML.s24Hour;
	
	DSLocalSystemTimeML.s12Hour;
	DSLocalSystemTimeML.sMin;
	DSLocalSystemTimeML.sSec;
	DSLocalSystemTimeML.s12HrSign;
	
	
	// SELECTED LANGUAGE
	eHmiLanguage;
	
	// Trigger ONE Scan Program
	acOneScan();
	
	

	// Get systen time from Beckhoff Function Block
	LocalSystemTime(
		sNetID:='' ,
		bEnable:=TRUE ,
		dwCycle:= ,
		dwOpt:= ,
		tTimeout:= ,
		bValid=> ,
		systemTime=>SysTime,
		tzID=> );
	
	sSysTime := TO_STRING(SYSTEMTIME_TO_DT(TIMESTR:= SysTime));
 	sSysTime := DELETE (sSysTime, 3,1);
		  
	(* Multi-Language*)
	// IF KEY IN WRONGLY ,OUT OF RANGE for selection
	IF eHmiLanguage < 1 THEN
	eHmiLanguage := 1;
	ELSIF eHmiLanguage > C_iLanguageQty THEN
	eHmiLanguage := C_iLanguageQty;
	END_IF
		
	
	// Manage the info to Data Structure
IF SysTime.wYear >2000 THEN
	acMultiLanguageControl();
END_IF

ACTION acMultiLanguageControl:
	// Push Info to DS - MULTILANGUAGE
	
		// sDayOfWeek, sMonth, s24Hour, s12Hour, s12HrSign
		DSLocalSystemTimeML.sDayOfWeek 	:= sLangDayOfWeek[eHmiLanguage,SysTime.wDayOfWeek];
		DSLocalSystemTimeML.sMonth 		:= sLangMonth[eHmiLanguage,SysTime.wMonth];
	
		IF SysTime.wHour < 10 THEN
		DSLocalSystemTimeML.s24Hour 	:= CONCAT ('0', WORD_TO_STRING(SysTime.wHour));
		ELSE
		DSLocalSystemTimeML.s24Hour  	:= WORD_TO_STRING(SysTime.wHour);
		END_IF
		
		IF SysTime.wHour = 0 THEN
		DSLocalSystemTimeML.s12Hour 	:= '12';
		DSLocalSystemTimeML.s12HrSign 	:= sLangAmPm[eHmiLanguage,1];
		
		ELSIF SysTime.wHour > 0 AND SysTime.wHour <12 THEN
		DSLocalSystemTimeML.s12Hour 	:= WORD_TO_STRING(SysTime.wHour);
		DSLocalSystemTimeML.s12HrSign 	:= sLangAmPm[eHmiLanguage,1];
		
		ELSIF SysTime.wHour > 0 AND SysTime.wHour =12 THEN
		DSLocalSystemTimeML.s12Hour 	:= WORD_TO_STRING(SysTime.wHour);
		DSLocalSystemTimeML.s12HrSign 	:= sLangAmPm[eHmiLanguage,2];
		
		ELSIF SysTime.wHour >= 13 THEN
		DSLocalSystemTimeML.s12Hour 	:= WORD_TO_STRING(SysTime.wHour-12);
		DSLocalSystemTimeML.s12HrSign 	:= sLangAmPm[eHmiLanguage,2];
		
		END_IF
	
		
		// sYear, sDay
		DSLocalSystemTimeML.sYear 		:= WORD_TO_STRING(SysTime.wYear);
		DSLocalSystemTimeML.sDay 		:= WORD_TO_STRING(SysTime.wDay);
	
		// sMin, sSec	
		IF SysTime.wMinute < 10 THEN
		DSLocalSystemTimeML.sMin 		:= CONCAT ('0', WORD_TO_STRING(SysTime.wMinute));
		ELSE
		DSLocalSystemTimeML.sMin 		:= WORD_TO_STRING(SysTime.wMinute);
		END_IF
		
		IF SysTime.wSecond < 10 THEN
		DSLocalSystemTimeML.sSec 		:= CONCAT ('0', WORD_TO_STRING(SysTime.wSecond));
		ELSE
		DSLocalSystemTimeML.sSec 		:= WORD_TO_STRING(SysTime.wSecond);
		END_IF
		

		// sCurrentDT12Hr

		DSLocalSystemTimeML.sCurrentDT12Hr  		:= CONCAT(DSLocalSystemTimeML.sDayOfWeek, ', ');
		DSLocalSystemTimeML.sCurrentDT12Hr  		:= CONCAT(DSLocalSystemTimeML.sCurrentDT12Hr, DSLocalSystemTimeML.sDay);
		DSLocalSystemTimeML.sCurrentDT12Hr  		:= CONCAT(DSLocalSystemTimeML.sCurrentDT12Hr, ' ');
		DSLocalSystemTimeML.sCurrentDT12Hr  		:= CONCAT(DSLocalSystemTimeML.sCurrentDT12Hr, DSLocalSystemTimeML.sMonth);
		DSLocalSystemTimeML.sCurrentDT12Hr  		:= CONCAT(DSLocalSystemTimeML.sCurrentDT12Hr, ' ');
		DSLocalSystemTimeML.sCurrentDT12Hr  		:= CONCAT(DSLocalSystemTimeML.sCurrentDT12Hr, DSLocalSystemTimeML.sYear);
		DSLocalSystemTimeML.sCurrentDT12Hr  		:= CONCAT(DSLocalSystemTimeML.sCurrentDT12Hr, ', ');
		DSLocalSystemTimeML.sCurrentDT12Hr  		:= CONCAT(DSLocalSystemTimeML.sCurrentDT12Hr, DSLocalSystemTimeML.s12Hour);
		DSLocalSystemTimeML.sCurrentDT12Hr  		:= CONCAT(DSLocalSystemTimeML.sCurrentDT12Hr, ':');
		DSLocalSystemTimeML.sCurrentDT12Hr  		:= CONCAT(DSLocalSystemTimeML.sCurrentDT12Hr, DSLocalSystemTimeML.sMin);
		DSLocalSystemTimeML.sCurrentDT12Hr  		:= CONCAT(DSLocalSystemTimeML.sCurrentDT12Hr, ':');
		DSLocalSystemTimeML.sCurrentDT12Hr  		:= CONCAT(DSLocalSystemTimeML.sCurrentDT12Hr, DSLocalSystemTimeML.sSec);
		DSLocalSystemTimeML.sCurrentDT12Hr  		:= CONCAT(DSLocalSystemTimeML.sCurrentDT12Hr, ' ');
		DSLocalSystemTimeML.sCurrentDT12Hr  		:= CONCAT(DSLocalSystemTimeML.sCurrentDT12Hr, DSLocalSystemTimeML.s12HrSign);


		// sCurrentDT24Hr

		DSLocalSystemTimeML.sCurrentDT24Hr  		:= CONCAT(DSLocalSystemTimeML.sDayOfWeek, ', ');
		DSLocalSystemTimeML.sCurrentDT24Hr  		:= CONCAT(DSLocalSystemTimeML.sCurrentDT24Hr, DSLocalSystemTimeML.sDay);
		DSLocalSystemTimeML.sCurrentDT24Hr  		:= CONCAT(DSLocalSystemTimeML.sCurrentDT24Hr, ' ');
		DSLocalSystemTimeML.sCurrentDT24Hr  		:= CONCAT(DSLocalSystemTimeML.sCurrentDT24Hr, DSLocalSystemTimeML.sMonth);
		DSLocalSystemTimeML.sCurrentDT24Hr  		:= CONCAT(DSLocalSystemTimeML.sCurrentDT24Hr, ' ');
		DSLocalSystemTimeML.sCurrentDT24Hr  		:= CONCAT(DSLocalSystemTimeML.sCurrentDT24Hr, DSLocalSystemTimeML.sYear);
		DSLocalSystemTimeML.sCurrentDT24Hr  		:= CONCAT(DSLocalSystemTimeML.sCurrentDT24Hr, ', ');
		DSLocalSystemTimeML.sCurrentDT24Hr  		:= CONCAT(DSLocalSystemTimeML.sCurrentDT24Hr, DSLocalSystemTimeML.s24Hour);
		DSLocalSystemTimeML.sCurrentDT24Hr  		:= CONCAT(DSLocalSystemTimeML.sCurrentDT24Hr, ':');
		DSLocalSystemTimeML.sCurrentDT24Hr  		:= CONCAT(DSLocalSystemTimeML.sCurrentDT24Hr, DSLocalSystemTimeML.sMin);
		DSLocalSystemTimeML.sCurrentDT24Hr  		:= CONCAT(DSLocalSystemTimeML.sCurrentDT24Hr, ':');
		DSLocalSystemTimeML.sCurrentDT24Hr  		:= CONCAT(DSLocalSystemTimeML.sCurrentDT24Hr, DSLocalSystemTimeML.sSec);

		// sCurrentDT24Hr_General
		
		DSLocalSystemTimeML.sCurrentDT24Hr_General  		:= CONCAT(DSLocalSystemTimeML.sDay, '/');
		DSLocalSystemTimeML.sCurrentDT24Hr_General  		:= CONCAT(DSLocalSystemTimeML.sCurrentDT24Hr_General, TO_STRING(SysTime.wMonth));
		DSLocalSystemTimeML.sCurrentDT24Hr_General  		:= CONCAT(DSLocalSystemTimeML.sCurrentDT24Hr_General, '/');
		DSLocalSystemTimeML.sCurrentDT24Hr_General  		:= CONCAT(DSLocalSystemTimeML.sCurrentDT24Hr_General, DSLocalSystemTimeML.sYear);
		DSLocalSystemTimeML.sCurrentDT24Hr_General  		:= CONCAT(DSLocalSystemTimeML.sCurrentDT24Hr_General, ' - ');
		DSLocalSystemTimeML.sCurrentDT24Hr_General  		:= CONCAT(DSLocalSystemTimeML.sCurrentDT24Hr_General, DSLocalSystemTimeML.s24Hour);
		DSLocalSystemTimeML.sCurrentDT24Hr_General  		:= CONCAT(DSLocalSystemTimeML.sCurrentDT24Hr_General, ':');
		DSLocalSystemTimeML.sCurrentDT24Hr_General  		:= CONCAT(DSLocalSystemTimeML.sCurrentDT24Hr_General, DSLocalSystemTimeML.sMin);
		DSLocalSystemTimeML.sCurrentDT24Hr_General  		:= CONCAT(DSLocalSystemTimeML.sCurrentDT24Hr_General, ':');
		DSLocalSystemTimeML.sCurrentDT24Hr_General  		:= CONCAT(DSLocalSystemTimeML.sCurrentDT24Hr_General, DSLocalSystemTimeML.sSec);

		// sCurrentDate_General
IF NOT bOverrideCurrentDate THEN
			// sYear & sMonth	
			IF SysTime.wMonth < 10 THEN
			DSLocalSystemTimeML.sCurrentDate_General 		:= CONCAT (WORD_TO_STRING(SysTime.wYear),'0');
			DSLocalSystemTimeML.sCurrentDate_General 		:= CONCAT (DSLocalSystemTimeML.sCurrentDate_General,WORD_TO_STRING(SysTime.wMonth));
			ELSE
			DSLocalSystemTimeML.sCurrentDate_General 		:= CONCAT (WORD_TO_STRING(SysTime.wYear),WORD_TO_STRING(SysTime.wMonth));
			END_IF

			// sDay	
			IF SysTime.wDay < 10 THEN
			DSLocalSystemTimeML.sCurrentDate_General 		:= CONCAT (DSLocalSystemTimeML.sCurrentDate_General,'0');
			DSLocalSystemTimeML.sCurrentDate_General 		:= CONCAT (DSLocalSystemTimeML.sCurrentDate_General,WORD_TO_STRING(SysTime.wDay));
			ELSE
			DSLocalSystemTimeML.sCurrentDate_General 		:= CONCAT (DSLocalSystemTimeML.sCurrentDate_General,WORD_TO_STRING(SysTime.wDay));
			END_IF
END_IF

		// sCurrentTime24Hr_General

			// sYear & sMonth	
			DSLocalSystemTimeML.sCurrentTime24Hr_General  	:= CONCAT(DSLocalSystemTimeML.sCurrentTime24Hr_General, DSLocalSystemTimeML.s24Hour);
			DSLocalSystemTimeML.sCurrentTime24Hr_General  	:= CONCAT(DSLocalSystemTimeML.sCurrentTime24Hr_General, ':');
			DSLocalSystemTimeML.sCurrentTime24Hr_General  	:= CONCAT(DSLocalSystemTimeML.sCurrentTime24Hr_General, DSLocalSystemTimeML.sMin);
			DSLocalSystemTimeML.sCurrentTime24Hr_General  	:= CONCAT(DSLocalSystemTimeML.sCurrentTime24Hr_General, ':');
			DSLocalSystemTimeML.sCurrentTime24Hr_General  	:= CONCAT(DSLocalSystemTimeML.sCurrentTime24Hr_General, DSLocalSystemTimeML.sSec);

		// dtCurrentDateTime
			DSLocalSystemTimeML.dtCurrentDateTime			:= SYSTEMTIME_TO_DT(SysTime);
		
		// sCurrentDateTime
			DSLocalSystemTimeML.sCurrentDateTime			:= DELETE(STR:= TO_STRING(DSLocalSystemTimeML.dtCurrentDateTime) , LEN:= 3, POS:= 1)		;
END_ACTION

ACTION acOneScan:

(*PREFIX Language*)
bOneScanRE(CLK:=TRUE , Q=> );

IF bOneScanRe.Q THEN

// ENGLISH
		
		(*DayOfWeek - English*)
		sLangDayOfWeek[1,1] := 'Mon';
		sLangDayOfWeek[1,2] := 'Tue';
		sLangDayOfWeek[1,3] := 'Wed';
		sLangDayOfWeek[1,4] := 'Thu';
		sLangDayOfWeek[1,5] := 'Fri';
		sLangDayOfWeek[1,6] := 'Sat';
		sLangDayOfWeek[1,0] := 'Sun';
		
		(*Month - English*)
		sLangMonth[1,1] := 'Jan';
		sLangMonth[1,2] := 'Feb';
		sLangMonth[1,3] := 'Mar';
		sLangMonth[1,4] := 'Apr';
		sLangMonth[1,5] := 'May';
		sLangMonth[1,6] := 'June';
		sLangMonth[1,7] := 'July';
		sLangMonth[1,8] := 'Aug';
		sLangMonth[1,9] := 'Sept';
		sLangMonth[1,10] := 'Oct';
		sLangMonth[1,11] := 'Nov';
		sLangMonth[1,12] := 'Dec';

		(*AmPm - English*)
		sLangAmPm[1,1] := 'AM';
		sLangAmPm[1,2] := 'PM';


		
// CHINESE
	
		(*DayOfWeek - Chinese*)
		sLangDayOfWeek[2,1] := '星期一';
		sLangDayOfWeek[2,2] := '星期二';
		sLangDayOfWeek[2,3] := '星期三';
		sLangDayOfWeek[2,4] := '星期四';
		sLangDayOfWeek[2,5] := '星期五';
		sLangDayOfWeek[2,6] := '星期六';
		sLangDayOfWeek[2,0] := '星期日';	
		
		(*Month - Chinese*)
		sLangMonth[2,1] := '一月';
		sLangMonth[2,2] := '二月';
		sLangMonth[2,3] := '三月';
		sLangMonth[2,4] := '四月';
		sLangMonth[2,5] := '五月';
		sLangMonth[2,6] := '六月';
		sLangMonth[2,7] := '七月';
		sLangMonth[2,8] := '八月';
		sLangMonth[2,9] := '九月';
		sLangMonth[2,10] := '十月';
		sLangMonth[2,11] := '十一月';
		sLangMonth[2,12] := '十二月';

		(*AmPm - Chinese*)
		sLangAmPm[2,1] := '早上';
		sLangAmPm[2,2] := '下午';
		
		
		
// GERMAN
		
		(*DayOfWeek - German*)
		sLangDayOfWeek[3,1] := 'Mon';
		sLangDayOfWeek[3,2] := 'Die';
		sLangDayOfWeek[3,3] := 'Mit';
		sLangDayOfWeek[3,4] := 'Don';
		sLangDayOfWeek[3,5] := 'Fre';
		sLangDayOfWeek[3,6] := 'Sam';
		sLangDayOfWeek[3,0] := 'Son';
		
		(*Month - German*)
		sLangMonth[3,1] := 'Jan';
		sLangMonth[3,2] := 'Feb';
		sLangMonth[3,3] := 'März';
		sLangMonth[3,4] := 'Apr';
		sLangMonth[3,5] := 'Mai';
		sLangMonth[3,6] := 'Juni';
		sLangMonth[3,7] := 'Juli';
		sLangMonth[3,8] := 'Aug';
		sLangMonth[3,9] := 'Sept';
		sLangMonth[3,10] := 'Okt';
		sLangMonth[3,11] := 'Nov';
		sLangMonth[3,12] := 'Dez';

		(*AmPm - German*)
		sLangAmPm[3,1] := 'AM';
		sLangAmPm[3,2] := 'PM';

		
// FRENCH

		(*DayOfWeek - French*)
		sLangDayOfWeek[4,1] := 'Lun';
		sLangDayOfWeek[4,2] := 'Mar';
		sLangDayOfWeek[4,3] := 'Mer';
		sLangDayOfWeek[4,4] := 'Jeu';
		sLangDayOfWeek[4,5] := 'Ven';
		sLangDayOfWeek[4,6] := 'Sam';
		sLangDayOfWeek[4,0] := 'Dim';
		
		(*Month - French*)
		sLangMonth[4,1] := 'Janv';
		sLangMonth[4,2] := 'Févr';
		sLangMonth[4,3] := 'Mars';
		sLangMonth[4,4] := 'Avril';
		sLangMonth[4,5] := 'Mai';
		sLangMonth[4,6] := 'Juin';
		sLangMonth[4,7] := 'Juil';
		sLangMonth[4,8] := 'Août';
		sLangMonth[4,9] := 'Sept';
		sLangMonth[4,10] := 'Oct';
		sLangMonth[4,11] := 'Nov';
		sLangMonth[4,12] := 'Déc';

		(*AmPm - French*)
		sLangAmPm[4,1] := 'AM';
		sLangAmPm[4,2] := 'PM';
	
	
// PORTUGUESE
		
		(*DayOfWeek - Portuguese*)
		sLangDayOfWeek[5,1] := 'Seg';
		sLangDayOfWeek[5,2] := 'Ter';
		sLangDayOfWeek[5,3] := 'Qua';
		sLangDayOfWeek[5,4] := 'Qui';
		sLangDayOfWeek[5,5] := 'Sex';
		sLangDayOfWeek[5,6] := 'Sáb';
		sLangDayOfWeek[5,0] := 'Dom';
		
		(*Month - Portuguese*)
		sLangMonth[5,1] := 'Jan';
		sLangMonth[5,2] := 'Fev';
		sLangMonth[5,3] := 'Março';
		sLangMonth[5,4] := 'Abril';
		sLangMonth[5,5] := 'Maio';
		sLangMonth[5,6] := 'Junho';
		sLangMonth[5,7] := 'Julho';
		sLangMonth[5,8] := 'Agosto';
		sLangMonth[5,9] := 'Set';
		sLangMonth[5,10] := 'Out';
		sLangMonth[5,11] := 'Nov';
		sLangMonth[5,12] := 'Dez';

		(*AmPm - Portuguese*)
		sLangAmPm[5,1] := 'AM';
		sLangAmPm[5,2] := 'PM';


END_IF
END_ACTION

END_PROGRAM

// ---- POUs/MainProgram/A_StandardStructureProgram/stUPSStatusMonitoring.TcPOU
PROGRAM stUPSStatusMonitoring
VAR
	fbGetUpsStatusfb: FB_GetUPSStatus;


END_VAR

fbGetUpsStatusfb(
	sNetId:= '',
	nPort:= 0,
	bEnable:= bGetUpsStatusEn,
	bValid=> bGetUpsStatusValid,
	bError=> bGetUpsStatusError,
	nErrId=> udiGetUpsStatusErrID,
	stStatus=> UpsStatus);

(* Check DC Power Status*)
IF UpsStatus.ePowerStatus = PowerUnknownStatus THEN
bDCPowerUnknownStatusAlarm := TRUE;
ELSE
bDCPowerUnknownStatusAlarm := FALSE;
END_IF

IF UpsStatus.ePowerStatus = PowerOnLine THEN
bDCPowerModeActivated := TRUE;
ELSE
bDCPowerModeActivated := FALSE;
END_IF

IF UpsStatus.ePowerStatus = PowerOnBattery THEN
bBatteryModeActivated := TRUE;
ELSE
bBatteryModeActivated := FALSE;
END_IF


(* Check Battery Status*)
IF UpsStatus.eBatteryStatus = BatteryUnknownStatus THEN
bBatteryUnknownStatusAlarm := TRUE;
ELSE
bBatteryUnknownStatusAlarm := FALSE;
END_IF

IF UpsStatus.eBatteryStatus = BatteryReplace THEN
bBatteryReplacementRequestAlarm := TRUE;
ELSE
bBatteryReplacementRequestAlarm := FALSE;
END_IF

(* Check UPS Comm Status *)
IF UpsStatus.eCommStatus = UpsCommUnknownStatus THEN
bUpsCommUnknownStatusAlarm := TRUE;
ELSE
bUpsCommUnknownStatusAlarm := FALSE;
END_IF

IF UpsStatus.eCommStatus = UpsCommOk THEN
bUpsCommOkFlag := TRUE;
ELSE
bUpsCommOkFlag := FALSE;
END_IF

IF UpsStatus.eCommStatus = UpsCommFailed THEN
bUpsCommErrorAlarm := TRUE;
ELSE
bUpsCommErrorAlarm := FALSE;
END_IF

END_PROGRAM

// ---- POUs/MainProgram/A_StandardStructureProgram/stWritePersistentData.TcPOU
PROGRAM stWritePersistentData
VAR
	AutoSaveTimer: TON;
	AutoSaveTimerRE: R_TRIG;
	tBackupDelayOnTimer: TON;
	BusyFE: F_TRIG;
	SaveDelayTimer: TON;
	SaveHR: BOOL;
	SaveDelayTimerRE: R_TRIG;
	fbWritePersistentData: FB_WritePersistentData;
	bManualWriteExecute: BOOL;
	bWritePDBusy: BOOL;
	bWritePDErr: BOOL;
	tAutoSaveTimerPV: TIME;
	tBackupDelayOffTimer: TON;
	bInternalPersistentBackup: BOOL;

END_VAR

IF bRecipeSavePb THEN
SaveHR := TRUE;
END_IF

AutoSaveTimer(IN:=NOT AutoSaveTimer.Q , PT:=t#10m , Q=> , ET=>tAutoSaveTimerPV );
AutoSaveTimerRE(CLK:=AutoSaveTimer.Q , Q=> );

SaveDelayTimer(IN:=SaveHR , PT:=T#2S , Q=> , ET=> );
SaveDelayTimerRE(CLK:=SaveDelayTimer.Q , Q=> );

IF SaveHR AND SaveDelayTimer.Q THEN
SaveHR := FALSE;
END_IF


fbWritePersistentData(
	NETID:= '' (*'5.38.239.218.1.1'*),
	PORT:=851 ,
	START:=AutoSaveTimerRE.Q OR SaveDelayTimerRE.Q OR bManualWriteExecute ,
	TMOUT:=t#10s ,
	MODE:=SPDM_VAR_BOOST ,
	BUSY=>bWritePDBusy ,
	ERR=>bWritePDErr ,
	ERRID=> );

(*Dr Yoges Data persistence backup*)
BusyFE(CLK:=bWritePDBusy , Q=> );

IF BusyFE.Q THEN
	bInternalPersistentBackup:=TRUE;
END_IF


tBackupDelayOnTimer(IN:=bInternalPersistentBackup , PT:=t#3s , Q=> , ET=> );
tBackupDelayOffTimer(IN:=tBackupDelayOnTimer.Q , PT:=t#0.5s , Q=> , ET=> );

IF tBackupDelayOnTimer.Q AND NOT tBackupDelayOffTimer.Q THEN
	silent_backup:=TRUE;
END_IF

IF tBackupDelayOffTimer.Q THEN
	silent_backup:=FALSE;
	bInternalPersistentBackup:=FALSE;
END_IF

END_PROGRAM

// ---- POUs/MainProgram/Aa_HmiVariableCtrl/HMIValueKeyInCtrl.TcPOU
PROGRAM HMIValueKeyInCtrl
VAR
	PowerOnDelayRE: R_TRIG;
END_VAR

(*OFF When using Indusoft HMI*)

(*xxxxxxxxxxxx 1st Visu Shown When Boot Up xxxxxxxxxxxx*)

PowerOnDelayRE(CLK:=PowerOnDelay.Q , Q=> );

IF PowerOnDelayRE.Q THEN
VisuElems.CurrentVisu := 'ZMAIN_PAGE' ;
END_IF


(*xxxxxxxxxxxx Station Process Time Display Monitoring - Pull out from Function Block xxxxxxxxxxxx*) (*Display ONLY*)
ARDsStnSeqProcessCtrl[1].In_AR5iCallTotalTimeRecipeNo[5] := DSStnBasketInfo[1].iStationSeqenceRecipeNo;
ARDsStnSeqProcessCtrl[2].In_AR5iCallTotalTimeRecipeNo[5] := DSStnBasketInfo[2].iStationSeqenceRecipeNo;
ARDsStnSeqProcessCtrl[3].In_AR5iCallTotalTimeRecipeNo[5] := DSStnBasketInfo[3].iStationSeqenceRecipeNo;
ARDsStnSeqProcessCtrl[4].In_AR5iCallTotalTimeRecipeNo[5] := DSStnBasketInfo[4].iStationSeqenceRecipeNo;
ARDsStnSeqProcessCtrl[5].In_AR5iCallTotalTimeRecipeNo[5] := DSStnBasketInfo[5].iStationSeqenceRecipeNo;
ARDsStnSeqProcessCtrl[6].In_AR5iCallTotalTimeRecipeNo[5] := DSStnBasketInfo[6].iStationSeqenceRecipeNo;
ARDsStnSeqProcessCtrl[7].In_AR5iCallTotalTimeRecipeNo[5] := DSStnBasketInfo[7].iStationSeqenceRecipeNo;
ARDsStnSeqProcessCtrl[8].In_AR5iCallTotalTimeRecipeNo[5] := DSStnBasketInfo[8].iStationSeqenceRecipeNo;
ARDsStnSeqProcessCtrl[9].In_AR5iCallTotalTimeRecipeNo[5] := DSStnBasketInfo[9].iStationSeqenceRecipeNo;
ARDsStnSeqProcessCtrl[10].In_AR5iCallTotalTimeRecipeNo[5] := DSStnBasketInfo[10].iStationSeqenceRecipeNo;
ARDsStnSeqProcessCtrl[11].In_AR5iCallTotalTimeRecipeNo[5] := DSStnBasketInfo[11].iStationSeqenceRecipeNo;
ARDsStnSeqProcessCtrl[12].In_AR5iCallTotalTimeRecipeNo[5] := DSStnBasketInfo[12].iStationSeqenceRecipeNo;

ARDsStnSeqProcessCtrl[1].Out_AR5iCalledTotalProcessTimeSV[5];
ARDsStnSeqProcessCtrl[2].Out_AR5iCalledTotalProcessTimeSV[5];
ARDsStnSeqProcessCtrl[3].Out_AR5iCalledTotalProcessTimeSV[5];
ARDsStnSeqProcessCtrl[4].Out_AR5iCalledTotalProcessTimeSV[5];
ARDsStnSeqProcessCtrl[5].Out_AR5iCalledTotalProcessTimeSV[5];
ARDsStnSeqProcessCtrl[6].Out_AR5iCalledTotalProcessTimeSV[5];
ARDsStnSeqProcessCtrl[7].Out_AR5iCalledTotalProcessTimeSV[5];
ARDsStnSeqProcessCtrl[8].Out_AR5iCalledTotalProcessTimeSV[5];
ARDsStnSeqProcessCtrl[9].Out_AR5iCalledTotalProcessTimeSV[5];
ARDsStnSeqProcessCtrl[10].Out_AR5iCalledTotalProcessTimeSV[5];
ARDsStnSeqProcessCtrl[11].Out_AR5iCalledTotalProcessTimeSV[5];
ARDsStnSeqProcessCtrl[12].Out_AR5iCalledTotalProcessTimeSV[5];


(*xxxxxxxxxxxx Temperature Ctrl xxxxxxxxxxxx*)

(*Station Temp Ctrl*)
	ARrStnTempHYSsv[1]; 			ARrStnTempHALsv[1]; 				ARrStnTempSV[1]; 			ARrStnTempRDYsv[1]; 			ARrStnTemp1stLimitSv[1];				ARrStnTemp2ndLimitSv[1];				ARiStnPreparationTempSv[1];
	ARrStnTempHYSsv[2]; 			ARrStnTempHALsv[2]; 				ARrStnTempSV[2]; 			ARrStnTempRDYsv[2];				ARrStnTemp1stLimitSv[2];				ARrStnTemp2ndLimitSv[2];				ARiStnPreparationTempSv[2];
	ARrStnTempHYSsv[3]; 			ARrStnTempHALsv[3]; 				ARrStnTempSV[3]; 			ARrStnTempRDYsv[3];				ARrStnTemp1stLimitSv[3];				ARrStnTemp2ndLimitSv[3];				ARiStnPreparationTempSv[3];
	ARrStnTempHYSsv[4]; 			ARrStnTempHALsv[4]; 				ARrStnTempSV[4]; 			ARrStnTempRDYsv[4];				ARrStnTemp1stLimitSv[4];				ARrStnTemp2ndLimitSv[4];				ARiStnPreparationTempSv[4];
	ARrStnTempHYSsv[5]; 			ARrStnTempHALsv[5]; 				ARrStnTempSV[5]; 			ARrStnTempRDYsv[5];				ARrStnTemp1stLimitSv[5];				ARrStnTemp2ndLimitSv[5];				ARiStnPreparationTempSv[5];
	ARrStnTempHYSsv[6]; 			ARrStnTempHALsv[6]; 				ARrStnTempSV[6]; 			ARrStnTempRDYsv[6];				ARrStnTemp1stLimitSv[6];				ARrStnTemp2ndLimitSv[6];				ARiStnPreparationTempSv[6];
	ARrStnTempHYSsv[7]; 			ARrStnTempHALsv[7]; 				ARrStnTempSV[7]; 			ARrStnTempRDYsv[7];				ARrStnTemp1stLimitSv[7];				ARrStnTemp2ndLimitSv[7];				ARiStnPreparationTempSv[7];
	ARrStnTempHYSsv[8]; 			ARrStnTempHALsv[8]; 				ARrStnTempSV[8]; 			ARrStnTempRDYsv[8];				ARrStnTemp1stLimitSv[8];				ARrStnTemp2ndLimitSv[8];				ARiStnPreparationTempSv[8];
	ARrStnTempHYSsv[9]; 			ARrStnTempHALsv[9]; 				ARrStnTempSV[9]; 			ARrStnTempRDYsv[9];				ARrStnTemp1stLimitSv[9];				ARrStnTemp2ndLimitSv[9];				ARiStnPreparationTempSv[9];
	ARrStnTempHYSsv[10]; 			ARrStnTempHALsv[10]; 			ARrStnTempSV[10]; 			ARrStnTempRDYsv[10];			ARrStnTemp1stLimitSv[10];				ARrStnTemp2ndLimitSv[10];			ARiStnPreparationTempSv[10];
	ARrStnTempHYSsv[11]; 			ARrStnTempHALsv[11]; 			ARrStnTempSV[11]; 			ARrStnTempRDYsv[11];			ARrStnTemp1stLimitSv[11];				ARrStnTemp2ndLimitSv[11];			ARiStnPreparationTempSv[11];
	ARrStnTempHYSsv[12]; 			ARrStnTempHALsv[12]; 			ARrStnTempSV[12]; 			ARrStnTempRDYsv[12];			ARrStnTemp1stLimitSv[12];				ARrStnTemp2ndLimitSv[12];			ARiStnPreparationTempSv[12];

(*Stn WaterJacket Temp Ctrl*)
	ARrStnWaterJacketTempHYSsv[4]; 	ARrStnWaterJacketTempHALsv[4]; 	ARrStnWaterJacketTempSV[4]; 	ARrStnWaterJacketTempRDYsv[4]; 	ARrStnWaterJacketTemp1stLimitSv[4]; 	ARrStnWaterJacketTemp2ndLimitSv[4]; 	ARiStnWaterJacketPreparationTempSv[4];
	ARrStnWaterJacketTempHYSsv[5]; 	ARrStnWaterJacketTempHALsv[5]; 	ARrStnWaterJacketTempSV[5]; 	ARrStnWaterJacketTempRDYsv[5]; 	ARrStnWaterJacketTemp1stLimitSv[5]; 	ARrStnWaterJacketTemp2ndLimitSv[5]; 	ARiStnWaterJacketPreparationTempSv[5];

(*Stn Sub Tank Temp Ctrl*)
	ARrStnSubTankTempHYSsv[1]; 			ARrStnSubTankTempHALsv[1]; 				ARrStnSubTankTempSV[1]; 			ARrStnSubTankTempRDYsv[1]; 			ARrStnSubTankTemp1stLimitSv[1];				ARrStnSubTankTemp2ndLimitSv[1];				ARiStnSubTankPreparationTempSv[1];
	ARrStnSubTankTempHYSsv[2]; 			ARrStnSubTankTempHALsv[2]; 				ARrStnSubTankTempSV[2]; 			ARrStnSubTankTempRDYsv[2];				ARrStnSubTankTemp1stLimitSv[2];				ARrStnSubTankTemp2ndLimitSv[2];				ARiStnSubTankPreparationTempSv[2];
	ARrStnSubTankTempHYSsv[3]; 			ARrStnSubTankTempHALsv[3]; 				ARrStnSubTankTempSV[3]; 			ARrStnSubTankTempRDYsv[3];				ARrStnSubTankTemp1stLimitSv[3];				ARrStnSubTankTemp2ndLimitSv[3];				ARiStnSubTankPreparationTempSv[3];
	ARrStnSubTankTempHYSsv[4]; 			ARrStnSubTankTempHALsv[4]; 				ARrStnSubTankTempSV[4]; 			ARrStnSubTankTempRDYsv[4];				ARrStnSubTankTemp1stLimitSv[4];				ARrStnSubTankTemp2ndLimitSv[4];				ARiStnSubTankPreparationTempSv[4];

(*JRS Inline Heater Temp Ctrl*)
	rJRSInlineHeaterTempHYSsv;
	rJRSInlineHeaterTempHALsv;
	rJRSInlineHeaterTempSV;
	rJRSInlineHeaterTempRDYsv;
	rJRSInlineHeaterTemp1stLimitSv;
	rJRSInlineHeaterTemp2ndLimitSv;
	iJRSInlineHeaterPreparationTempSv	;

(*Inc Temp Ctrl*)
	rIncTempHYSsv;
	rIncTempHALsv;
	rIncTempSV;
	rIncTempRDYsv;
	rIncTemp1stLimitSv;
	rIncTemp2ndLimitSv;
	iIncPreparationTempSv;

(*Oil Separator Temp Ctrl*)
	rOilSeparatorTempHYSsv;
	rOilSeparatorTempHALsv;
	rOilSeparatorTempSV;
	rOilSeparatorTempRDYsv;
	rOilSeparatorTemp1stLimitSv;
	rOilSeparatorTemp2ndLimitSv;
	iOilSeparatorPreparationTempSv;


(*xxxxxxxxxxxx Conductivity Setting  xxxxxxxxxxxx*)

(*1st/2nd Limit - Use this as the setting when the tank is using DI water/Normal water*)
	ARrStnConductivity1stLimitSv[1]; 			ARrStnConductivity2ndLimitSv[1];
	ARrStnConductivity1stLimitSv[2]; 			ARrStnConductivity2ndLimitSv[2];
	ARrStnConductivity1stLimitSv[3]; 			ARrStnConductivity2ndLimitSv[3];
	ARrStnConductivity1stLimitSv[4]; 			ARrStnConductivity2ndLimitSv[4];
	ARrStnConductivity1stLimitSv[5]; 			ARrStnConductivity2ndLimitSv[5];
	ARrStnConductivity1stLimitSv[6]; 			ARrStnConductivity2ndLimitSv[6];
	ARrStnConductivity1stLimitSv[7]; 			ARrStnConductivity2ndLimitSv[7];
	ARrStnConductivity1stLimitSv[8]; 			ARrStnConductivity2ndLimitSv[8];
	ARrStnConductivity1stLimitSv[9]; 			ARrStnConductivity2ndLimitSv[9];
	ARrStnConductivity1stLimitSv[10]; 		ARrStnConductivity2ndLimitSv[10];
	ARrStnConductivity1stLimitSv[11]; 		ARrStnConductivity2ndLimitSv[11];
	ARrStnConductivity1stLimitSv[12]; 		ARrStnConductivity2ndLimitSv[12];

(*Low/High - Use this as the setting when the tank is using Chemical/Detergent*)
	ARrStnLowConductivitySv[1]; 			ARrStnHighConductivitySv[1];
	ARrStnLowConductivitySv[2]; 			ARrStnHighConductivitySv[2];
	ARrStnLowConductivitySv[3]; 			ARrStnHighConductivitySv[3];
	ARrStnLowConductivitySv[4]; 			ARrStnHighConductivitySv[4];
	ARrStnLowConductivitySv[5]; 			ARrStnHighConductivitySv[5];
	ARrStnLowConductivitySv[6]; 			ARrStnHighConductivitySv[6];
	ARrStnLowConductivitySv[7]; 			ARrStnHighConductivitySv[7];
	ARrStnLowConductivitySv[8]; 			ARrStnHighConductivitySv[8];
	ARrStnLowConductivitySv[9]; 			ARrStnHighConductivitySv[9];
	ARrStnLowConductivitySv[10]; 			ARrStnHighConductivitySv[10];
	ARrStnLowConductivitySv[11]; 			ARrStnHighConductivitySv[11];
	ARrStnLowConductivitySv[12]; 			ARrStnHighConductivitySv[12];


(*xxxxxxxxxxxx Resistivity Setting  xxxxxxxxxxxx*)

(*1st/2nd Limit - Use this as the setting when the tank is using DI water/Normal water*)
(*	ARrStnResistivity1stLimitSv[1]; 			ARrStnResistivity2ndLimitSv[1];
	ARrStnResistivity1stLimitSv[2]; 			ARrStnResistivity2ndLimitSv[2];
	ARrStnResistivity1stLimitSv[3]; 			ARrStnResistivity2ndLimitSv[3];
	ARrStnResistivity1stLimitSv[4]; 			ARrStnResistivity2ndLimitSv[4];
	ARrStnResistivity1stLimitSv[5]; 			ARrStnResistivity2ndLimitSv[5];
	ARrStnResistivity1stLimitSv[6]; 			ARrStnResistivity2ndLimitSv[6];
	ARrStnResistivity1stLimitSv[7]; 			ARrStnResistivity2ndLimitSv[7];
	ARrStnResistivity1stLimitSv[8]; 			ARrStnResistivity2ndLimitSv[8];
	ARrStnResistivity1stLimitSv[9]; 			ARrStnResistivity2ndLimitSv[9];
	ARrStnResistivity1stLimitSv[10]; 			ARrStnResistivity2ndLimitSv[10];
	ARrStnResistivity1stLimitSv[11]; 			ARrStnResistivity2ndLimitSv[11];
	ARrStnResistivity1stLimitSv[12]; 			ARrStnResistivity2ndLimitSv[12];

(*Low/High - Use this as the setting when the tank is using Chemical/Detergent*)
	ARrStnLowResistivitySv[1]; 				ARrStnHighResistivitySv[1];
	ARrStnLowResistivitySv[2]; 				ARrStnHighResistivitySv[2];
	ARrStnLowResistivitySv[3]; 				ARrStnHighResistivitySv[3];
	ARrStnLowResistivitySv[4]; 				ARrStnHighResistivitySv[4];
	ARrStnLowResistivitySv[5]; 				ARrStnHighResistivitySv[5];
	ARrStnLowResistivitySv[6]; 				ARrStnHighResistivitySv[6];
	ARrStnLowResistivitySv[7]; 				ARrStnHighResistivitySv[7];
	ARrStnLowResistivitySv[8]; 				ARrStnHighResistivitySv[8];
	ARrStnLowResistivitySv[9]; 				ARrStnHighResistivitySv[9];
	ARrStnLowResistivitySv[10]; 			ARrStnHighResistivitySv[10];
	ARrStnLowResistivitySv[11]; 			ARrStnHighResistivitySv[11];
	ARrStnLowResistivitySv[12]; 			ARrStnHighResistivitySv[12];


(*xxxxxxxxxxxx PH Setting  xxxxxxxxxxxx*)

(*Low/High*)
	ARrStnLowPhSv[1]; 					ARrStnHighPhSv[1];
	ARrStnLowPhSv[2]; 					ARrStnHighPhSv[2];
	ARrStnLowPhSv[3]; 					ARrStnHighPhSv[3];
	ARrStnLowPhSv[4]; 					ARrStnHighPhSv[4];
	ARrStnLowPhSv[5]; 					ARrStnHighPhSv[5];
	ARrStnLowPhSv[6]; 					ARrStnHighPhSv[6];
	ARrStnLowPhSv[7]; 					ARrStnHighPhSv[7];
	ARrStnLowPhSv[8]; 					ARrStnHighPhSv[8];
	ARrStnLowPhSv[9]; 					ARrStnHighPhSv[9];
	ARrStnLowPhSv[10]; 					ARrStnHighPhSv[10];
	ARrStnLowPhSv[11]; 					ARrStnHighPhSv[11];
	ARrStnLowPhSv[12]; 					ARrStnHighPhSv[12];
*)

(*xxxxxxxxxxxx Filter Pressure Setting  xxxxxxxxxxxx*)

(*1st/2nd Limit*)
	ARrStnFilterPressure1stLimitSv[1]; 		ARrStnFilterPressure2ndLimitSv[1];
	ARrStnFilterPressure1stLimitSv[2]; 		ARrStnFilterPressure2ndLimitSv[2];
	ARrStnFilterPressure1stLimitSv[3]; 		ARrStnFilterPressure2ndLimitSv[3];
	ARrStnFilterPressure1stLimitSv[4]; 		ARrStnFilterPressure2ndLimitSv[4];
	ARrStnFilterPressure1stLimitSv[5]; 		ARrStnFilterPressure2ndLimitSv[5];
	ARrStnFilterPressure1stLimitSv[6]; 		ARrStnFilterPressure2ndLimitSv[6];
	ARrStnFilterPressure1stLimitSv[7]; 		ARrStnFilterPressure2ndLimitSv[7];
	ARrStnFilterPressure1stLimitSv[8]; 		ARrStnFilterPressure2ndLimitSv[8];
	ARrStnFilterPressure1stLimitSv[9]; 		ARrStnFilterPressure2ndLimitSv[9];
	ARrStnFilterPressure1stLimitSv[10]; 		ARrStnFilterPressure2ndLimitSv[10];
	ARrStnFilterPressure1stLimitSv[11]; 		ARrStnFilterPressure2ndLimitSv[11];
	ARrStnFilterPressure1stLimitSv[12]; 		ARrStnFilterPressure2ndLimitSv[12];


(*xxxxxxxxxxxx Flow Switch Setting  xxxxxxxxxxxx*)

(*1st/2nd Limit*)
	ARrStnFlowSwitch1stLimitSv[1]; 			ARrStnFlowSwitch2ndLimitSv[1];
	ARrStnFlowSwitch1stLimitSv[2]; 			ARrStnFlowSwitch2ndLimitSv[2];
	ARrStnFlowSwitch1stLimitSv[3]; 			ARrStnFlowSwitch2ndLimitSv[3];
	ARrStnFlowSwitch1stLimitSv[4]; 			ARrStnFlowSwitch2ndLimitSv[4];
	ARrStnFlowSwitch1stLimitSv[5]; 			ARrStnFlowSwitch2ndLimitSv[5];
	ARrStnFlowSwitch1stLimitSv[6]; 			ARrStnFlowSwitch2ndLimitSv[6];
	ARrStnFlowSwitch1stLimitSv[7]; 			ARrStnFlowSwitch2ndLimitSv[7];
	ARrStnFlowSwitch1stLimitSv[8]; 			ARrStnFlowSwitch2ndLimitSv[8];
	ARrStnFlowSwitch1stLimitSv[9]; 			ARrStnFlowSwitch2ndLimitSv[9];
	ARrStnFlowSwitch1stLimitSv[10]; 		ARrStnFlowSwitch2ndLimitSv[10];
	ARrStnFlowSwitch1stLimitSv[11]; 		ARrStnFlowSwitch2ndLimitSv[11];
	ARrStnFlowSwitch1stLimitSv[12]; 		ARrStnFlowSwitch2ndLimitSv[12];


(*xxxxxxxxxxxx Weber/Clangsonic Ultrasonic Power Setting - Manual Mode xxxxxxxxxxxx*)

(*Side Ultrasonic*)
	ARiStnManualUSSideAsv[1]; 			ARiStnManualUSSideBsv[1]; 			ARiStnManualUSSideCsv[1]; 			ARiStnManualUSSideDsv[1];
	ARiStnManualUSSideAsv[2]; 			ARiStnManualUSSideBsv[2]; 			ARiStnManualUSSideCsv[2]; 			ARiStnManualUSSideDsv[2];
	ARiStnManualUSSideAsv[3]; 			ARiStnManualUSSideBsv[3]; 			ARiStnManualUSSideCsv[3]; 			ARiStnManualUSSideDsv[3];
	ARiStnManualUSSideAsv[4]; 			ARiStnManualUSSideBsv[4]; 			ARiStnManualUSSideCsv[4]; 			ARiStnManualUSSideDsv[4];
	ARiStnManualUSSideAsv[5]; 			ARiStnManualUSSideBsv[5]; 			ARiStnManualUSSideCsv[5]; 			ARiStnManualUSSideDsv[5];
	ARiStnManualUSSideAsv[6]; 			ARiStnManualUSSideBsv[6]; 			ARiStnManualUSSideCsv[6]; 			ARiStnManualUSSideDsv[6];
	ARiStnManualUSSideAsv[7]; 			ARiStnManualUSSideBsv[7]; 			ARiStnManualUSSideCsv[7]; 			ARiStnManualUSSideDsv[7];
	ARiStnManualUSSideAsv[8]; 			ARiStnManualUSSideBsv[8]; 			ARiStnManualUSSideCsv[8]; 			ARiStnManualUSSideDsv[8];
	ARiStnManualUSSideAsv[9]; 			ARiStnManualUSSideBsv[9]; 			ARiStnManualUSSideCsv[9]; 			ARiStnManualUSSideDsv[9];
	ARiStnManualUSSideAsv[10]; 			ARiStnManualUSSideBsv[10]; 			ARiStnManualUSSideCsv[10]; 			ARiStnManualUSSideDsv[10];
	ARiStnManualUSSideAsv[11]; 			ARiStnManualUSSideBsv[11]; 			ARiStnManualUSSideCsv[11]; 			ARiStnManualUSSideDsv[11];
	ARiStnManualUSSideAsv[12]; 			ARiStnManualUSSideBsv[12]; 			ARiStnManualUSSideCsv[12]; 			ARiStnManualUSSideDsv[12];

(*Bottom Ultrasonic*)
	ARiStnManualUSBtmAsv[1]; 			ARiStnManualUSBtmBsv[1]; 			ARiStnManualUSBtmCsv[1]; 			ARiStnManualUSBtmDsv[1];
	ARiStnManualUSBtmAsv[2]; 			ARiStnManualUSBtmBsv[2]; 			ARiStnManualUSBtmCsv[2]; 			ARiStnManualUSBtmDsv[2];
	ARiStnManualUSBtmAsv[3]; 			ARiStnManualUSBtmBsv[3]; 			ARiStnManualUSBtmCsv[3]; 			ARiStnManualUSBtmDsv[3];
	ARiStnManualUSBtmAsv[4]; 			ARiStnManualUSBtmBsv[4]; 			ARiStnManualUSBtmCsv[4]; 			ARiStnManualUSBtmDsv[4];
	ARiStnManualUSBtmAsv[5]; 			ARiStnManualUSBtmBsv[5]; 			ARiStnManualUSBtmCsv[5]; 			ARiStnManualUSBtmDsv[5];
	ARiStnManualUSBtmAsv[6]; 			ARiStnManualUSBtmBsv[6]; 			ARiStnManualUSBtmCsv[6]; 			ARiStnManualUSBtmDsv[6];
	ARiStnManualUSBtmAsv[7]; 			ARiStnManualUSBtmBsv[7]; 			ARiStnManualUSBtmCsv[7]; 			ARiStnManualUSBtmDsv[7];
	ARiStnManualUSBtmAsv[8]; 			ARiStnManualUSBtmBsv[8]; 			ARiStnManualUSBtmCsv[8]; 			ARiStnManualUSBtmDsv[8];
	ARiStnManualUSBtmAsv[9]; 			ARiStnManualUSBtmBsv[9]; 			ARiStnManualUSBtmCsv[9]; 			ARiStnManualUSBtmDsv[9];
	ARiStnManualUSBtmAsv[10]; 			ARiStnManualUSBtmBsv[10]; 			ARiStnManualUSBtmCsv[10]; 			ARiStnManualUSBtmDsv[10];
	ARiStnManualUSBtmAsv[11]; 			ARiStnManualUSBtmBsv[11]; 			ARiStnManualUSBtmCsv[11]; 			ARiStnManualUSBtmDsv[11];
	ARiStnManualUSBtmAsv[12]; 			ARiStnManualUSBtmBsv[12]; 			ARiStnManualUSBtmCsv[12]; 			ARiStnManualUSBtmDsv[12];


(*xxxxxxxxxxxx Vacuum Setting  xxxxxxxxxxxx*)

(*Stn Vacuum High/Low Level*)
(*	ARrStnHighVacuumLevelSV[1]; 			ARrStnLowVacuumLevelSV[1];
	ARrStnHighVacuumLevelSV[2]; 			ARrStnLowVacuumLevelSV[2];
	ARrStnHighVacuumLevelSV[3]; 			ARrStnLowVacuumLevelSV[3];
	ARrStnHighVacuumLevelSV[4]; 			ARrStnLowVacuumLevelSV[4];
	ARrStnHighVacuumLevelSV[5]; 			ARrStnLowVacuumLevelSV[5];
	ARrStnHighVacuumLevelSV[6]; 			ARrStnLowVacuumLevelSV[6];
	ARrStnHighVacuumLevelSV[7]; 			ARrStnLowVacuumLevelSV[7];
	ARrStnHighVacuumLevelSV[8]; 			ARrStnLowVacuumLevelSV[8];
	ARrStnHighVacuumLevelSV[9]; 			ARrStnLowVacuumLevelSV[9];
	ARrStnHighVacuumLevelSV[10]; 		ARrStnLowVacuumLevelSV[10];
	ARrStnHighVacuumLevelSV[11]; 		ARrStnLowVacuumLevelSV[11];
	ARrStnHighVacuumLevelSV[12]; 		ARrStnLowVacuumLevelSV[12];

(*Stn Sub Vacuum High/Low Level*)
	ARrStnSubHighVacuumLevelSV[1]; 		ARrStnSubLowVacuumLevelSV[1];
	ARrStnSubHighVacuumLevelSV[2]; 		ARrStnSubLowVacuumLevelSV[2];
	ARrStnSubHighVacuumLevelSV[3]; 		ARrStnSubLowVacuumLevelSV[3];
	ARrStnSubHighVacuumLevelSV[4]; 		ARrStnSubLowVacuumLevelSV[4];
	ARrStnSubHighVacuumLevelSV[5]; 		ARrStnSubLowVacuumLevelSV[5];
	ARrStnSubHighVacuumLevelSV[6]; 		ARrStnSubLowVacuumLevelSV[6];
	ARrStnSubHighVacuumLevelSV[7]; 		ARrStnSubLowVacuumLevelSV[7];
	ARrStnSubHighVacuumLevelSV[8]; 		ARrStnSubLowVacuumLevelSV[8];
	ARrStnSubHighVacuumLevelSV[9]; 		ARrStnSubLowVacuumLevelSV[9];
	ARrStnSubHighVacuumLevelSV[10]; 		ARrStnSubLowVacuumLevelSV[10];
	ARrStnSubHighVacuumLevelSV[11]; 		ARrStnSubLowVacuumLevelSV[11];
	ARrStnSubHighVacuumLevelSV[12]; 		ARrStnSubLowVacuumLevelSV[12];

(*DC/CC Vacuum High/Low Level*)
	rDCHighVacuumLevelSV; 				ARrCCHighVacuumLevelSV[4];		ARrCCHighVacuumLevelSV[5];
	rDCLowVacuumLevelSV; 				ARrCCLowVacuumLevelSV[4];		ARrCCLowVacuumLevelSV[5];

(*Rev Vacuum High/Low Level*)
	ARrRevHighVacuumLevelSV[1]; 		ARrRevLowVacuumLevelSV[1];
	ARrRevHighVacuumLevelSV[2]; 		ARrRevLowVacuumLevelSV[2];
	ARrRevHighVacuumLevelSV[3]; 		ARrRevLowVacuumLevelSV[3];
	ARrRevHighVacuumLevelSV[4]; 		ARrRevLowVacuumLevelSV[4];
	ARrRevHighVacuumLevelSV[5]; 		ARrRevLowVacuumLevelSV[5];
	ARrRevHighVacuumLevelSV[6]; 		ARrRevLowVacuumLevelSV[6];
	ARrRevHighVacuumLevelSV[7]; 		ARrRevLowVacuumLevelSV[7];
	ARrRevHighVacuumLevelSV[8]; 		ARrRevLowVacuumLevelSV[8];
	ARrRevHighVacuumLevelSV[9]; 		ARrRevLowVacuumLevelSV[9];
	ARrRevHighVacuumLevelSV[10]; 		ARrRevLowVacuumLevelSV[10];
	ARrRevHighVacuumLevelSV[11]; 		ARrRevLowVacuumLevelSV[11];
	ARrRevHighVacuumLevelSV[12]; 		ARrRevLowVacuumLevelSV[12];

(*Stn Vacuum MaxRead SV*)
	ARlrStnVacuumMaxReadSV[1];
	ARlrStnVacuumMaxReadSV[2];
	ARlrStnVacuumMaxReadSV[3];
	ARlrStnVacuumMaxReadSV[4];
	ARlrStnVacuumMaxReadSV[5];
	ARlrStnVacuumMaxReadSV[6];
	ARlrStnVacuumMaxReadSV[7];
	ARlrStnVacuumMaxReadSV[8];
	ARlrStnVacuumMaxReadSV[9];
	ARlrStnVacuumMaxReadSV[10];
	ARlrStnVacuumMaxReadSV[11];
	ARlrStnVacuumMaxReadSV[12];

(*Stn Sub Vacuum MaxRead SV*)
	ARlrStnSubVacuumMaxReadSV[1];
	ARlrStnSubVacuumMaxReadSV[2];
	ARlrStnSubVacuumMaxReadSV[3];
	ARlrStnSubVacuumMaxReadSV[4];
	ARlrStnSubVacuumMaxReadSV[5];
	ARlrStnSubVacuumMaxReadSV[6];
	ARlrStnSubVacuumMaxReadSV[7];
	ARlrStnSubVacuumMaxReadSV[8];
	ARlrStnSubVacuumMaxReadSV[9];
	ARlrStnSubVacuumMaxReadSV[10];
	ARlrStnSubVacuumMaxReadSV[11];
	ARlrStnSubVacuumMaxReadSV[12];

(*DC/CC Vacuum MaxRead SV*)
	lrDCVacuumMaxReadSV;
	ARlrCCVacuumMaxReadSV[4];
	ARlrCCVacuumMaxReadSV[5];

(*Rev Vacuum MaxRead SV*)
	ARlrRevVacuumMaxReadSV[1];
	ARlrRevVacuumMaxReadSV[2];
	ARlrRevVacuumMaxReadSV[3];
	ARlrRevVacuumMaxReadSV[4];
	ARlrRevVacuumMaxReadSV[5];
	ARlrRevVacuumMaxReadSV[6];
	ARlrRevVacuumMaxReadSV[7];
	ARlrRevVacuumMaxReadSV[8];
	ARlrRevVacuumMaxReadSV[9];
	ARlrRevVacuumMaxReadSV[10];
	ARlrRevVacuumMaxReadSV[11];
	ARlrRevVacuumMaxReadSV[12];

*)
(*Stn Agitation DelayOffTimer SV*)
	iStnAgitation1DelayOffTimerSV_min;


(*xxxxxxxxxxxx Arm & Loading & Unloading Station ID xxxxxxxxxxxx*)
	ARiLdStnID[1]																	:= 79;
	ARiUldStnID[1]																	:= 81;
	(*ARiUldStnID[2];*)

	ARiArmID[1]																		:= 91;
	ARiArmID[2]																		:= 92;

	DSA1fbPnpSequenceMemoryStore.DsA1inPnpSequenceMemory.iLdGroupNo 				:= 1;
	DSA1fbPnpSequenceMemoryStore.DsA1inPnpSequenceMemory.iUldGroupNo 			:= 1;

	LdDSStationSSERStore.DsStationSequenceRecipeMemory.AR10iStationSubProNo[1]              := 1;
	LdDSStationSSURStore.DsSubRecipeMemory.bStCon19ExternalActivation				:= TRUE;


(*xxxxxxxxxxxx Arm Horz Zone Confirm Variable Ctrl xxxxxxxxxxxx*)

(*ARM 1*)
	ARlrArmHorzStartPoint[1]															:= 0;
	ARlrArmHorzEndPoint[1]															:= 10000;

	ARiArm1HorzListing[1]																:= 79; (*AR50*)
	ARiArm1HorzListing[2]																:= 1; (*AR50*)
	ARiArm1HorzListing[3]																:= 2; (*AR50*)
	ARiArm1HorzListing[4]																:= 3; (*AR50*)
	ARiArm1HorzListing[5]																:= 4; (*AR50*)
	ARiArm1HorzListing[6]																:= 5; (*AR50*)
	ARiArm1HorzListing[7]																:= 6; (*AR50*)
	ARiArm1HorzListing[8]																:= 7; (*AR50*)
	ARiArm1HorzListing[9]																:= 8; (*AR50*)
	ARiArm1HorzListing[10]															:= 9; (*AR50*)
	ARiArm1HorzListing[11]															:= 10; (*AR50*)
	ARiArm1HorzListing[12]															:= 81; (*AR50*)
	ARiArm1HorzListing[13]															:= 0; (*AR50*)
	ARiArm1HorzListing[14]															:= 0; (*AR50*)
	ARiArm1HorzListing[15]															:= 0; (*AR50*)

(*
(*ARM 2*)
	ARlrArmHorzStartPoint[2]															:= 0;
	ARlrArmHorzEndPoint[2]															:= 10000;

	ARiArm2HorzListing[1]																:= 81; (*AR50*)
	ARiArm2HorzListing[2]																:= 10; (*AR50*)
	ARiArm2HorzListing[3]																:= 9; (*AR50*)
	ARiArm2HorzListing[4]																:= 8; (*AR50*)
	ARiArm2HorzListing[5]																:= 7; (*AR50*)
	ARiArm2HorzListing[6]																:= 6; (*AR50*)
	ARiArm2HorzListing[7]																:= 0; (*AR50*)
	ARiArm2HorzListing[8]																:= 0; (*AR50*)
	ARiArm2HorzListing[9]																:= 0; (*AR50*)
	ARiArm2HorzListing[10]															:= 0; (*AR50*)
	ARiArm2HorzListing[11]															:= 0; (*AR50*)
	ARiArm2HorzListing[12]															:= 0; (*AR50*)
	ARiArm2HorzListing[13]															:= 0; (*AR50*)
	ARiArm2HorzListing[14]															:= 0; (*AR50*)
	ARiArm2HorzListing[15]															:= 0; (*AR50*)
*)

(*ARM 1*)
(*Station Hook, Unhook, Top, Bottom Position - from Beckhoff HMI*)
	Arm1HookPos[19]; (*Loading*)		Arm1UnHookPos[19]; 			Arm1TopPos[19]; 			Arm1BottomPos[19];
	Arm1HookPos[20]; (*Unloading*)		Arm1UnHookPos[20]; 			Arm1TopPos[20]; 			Arm1BottomPos[20];
	Arm1HookPos[1]; (*Station*)			Arm1UnHookPos[1]; 			Arm1TopPos[1]; 				Arm1BottomPos[1];
	Arm1HookPos[2];						Arm1UnHookPos[2]; 			Arm1TopPos[2]; 				Arm1BottomPos[2];
	Arm1HookPos[3];						Arm1UnHookPos[3]; 			Arm1TopPos[3]; 				Arm1BottomPos[3];
	Arm1HookPos[4];						Arm1UnHookPos[4]; 			Arm1TopPos[4]; 				Arm1BottomPos[4];
	Arm1HookPos[5]; 					Arm1UnHookPos[5]; 			Arm1TopPos[5]; 				Arm1BottomPos[5];
	Arm1HookPos[6]; 					Arm1UnHookPos[6]; 			Arm1TopPos[6]; 				Arm1BottomPos[6];
	Arm1HookPos[7]; 					Arm1UnHookPos[7]; 			Arm1TopPos[7]; 				Arm1BottomPos[7];
	Arm1HookPos[8]; 					Arm1UnHookPos[8]; 			Arm1TopPos[8]; 				Arm1BottomPos[8];
	Arm1HookPos[9]; 					Arm1UnHookPos[9]; 			Arm1TopPos[9]; 				Arm1BottomPos[9];
	Arm1HookPos[10]; 					Arm1UnHookPos[10]; 			Arm1TopPos[10]; 			Arm1BottomPos[10];
	Arm1HookPos[11]; 					Arm1UnHookPos[11]; 			Arm1TopPos[11]; 			Arm1BottomPos[11];
	Arm1HookPos[12]; 					Arm1UnHookPos[12]; 			Arm1TopPos[12]; 			Arm1BottomPos[12];

(*ARM 2*)
(*Station Hook, Unhook, Top, Bottom Position - from Beckhoff HMI*)
	Arm2HookPos[19]; (*Loading*)		Arm2UnHookPos[19]; 			Arm2TopPos[19]; 			Arm2BottomPos[19];
	Arm2HookPos[20]; (*Unloading*)		Arm2UnHookPos[20]; 			Arm2TopPos[20]; 			Arm2BottomPos[20];
	Arm2HookPos[1]; (*Station*)			Arm2UnHookPos[1]; 			Arm2TopPos[1]; 				Arm2BottomPos[1];
	Arm2HookPos[2];						Arm2UnHookPos[2]; 			Arm2TopPos[2]; 				Arm2BottomPos[2];
	Arm2HookPos[3];						Arm2UnHookPos[3]; 			Arm2TopPos[3]; 				Arm2BottomPos[3];
	Arm2HookPos[4];						Arm2UnHookPos[4]; 			Arm2TopPos[4]; 				Arm2BottomPos[4];
	Arm2HookPos[5]; 					Arm2UnHookPos[5]; 			Arm2TopPos[5]; 				Arm2BottomPos[5];
	Arm2HookPos[6]; 					Arm2UnHookPos[6]; 			Arm2TopPos[6]; 				Arm2BottomPos[6];
	Arm2HookPos[7]; 					Arm2UnHookPos[7]; 			Arm2TopPos[7]; 				Arm2BottomPos[7];
	Arm2HookPos[8]; 					Arm2UnHookPos[8]; 			Arm2TopPos[8]; 				Arm2BottomPos[8];
	Arm2HookPos[9]; 					Arm2UnHookPos[9]; 			Arm2TopPos[9]; 				Arm2BottomPos[9];
	Arm2HookPos[10]; 					Arm2UnHookPos[10]; 			Arm2TopPos[10]; 			Arm2BottomPos[10];
	Arm2HookPos[11]; 					Arm2UnHookPos[11]; 			Arm2TopPos[11]; 			Arm2BottomPos[11];
	Arm2HookPos[12]; 					Arm2UnHookPos[12]; 			Arm2TopPos[12]; 			Arm2BottomPos[12];


(*Station Hook Postion*)
(*ARM 1*)
	ARDSArmCtrl[1].AR3slrPosition[2,1,8];

	ARDSArmCtrl[1].AR3slrPosition[3,1,8];
	(*ARDSArmCtrl[1].AR3slrPosition[3,1,8];*)

	ARDSArmCtrl[1].AR3slrPosition[1,1,8];
	ARDSArmCtrl[1].AR3slrPosition[1,2,8];
	ARDSArmCtrl[1].AR3slrPosition[1,3,8];
	ARDSArmCtrl[1].AR3slrPosition[1,4,8];
	ARDSArmCtrl[1].AR3slrPosition[1,5,8];
	ARDSArmCtrl[1].AR3slrPosition[1,6,8];
	ARDSArmCtrl[1].AR3slrPosition[1,7,8];
	ARDSArmCtrl[1].AR3slrPosition[1,8,8];
	ARDSArmCtrl[1].AR3slrPosition[1,9,8];
	ARDSArmCtrl[1].AR3slrPosition[1,10,8];
	ARDSArmCtrl[1].AR3slrPosition[1,11,8];
	ARDSArmCtrl[1].AR3slrPosition[1,12,8];

(*On when using beckhoff HMI, Off when using Indusoft*)
(*ARM 1*)

	ARDSArmCtrl[1].AR3slrPosition[2,1,8]													:= Arm1HookPos[19];

	ARDSArmCtrl[1].AR3slrPosition[3,1,8]													:= Arm1HookPos[20];
	(*ARDSArmCtrl[1].AR3slrPosition[3,1,8];*)

	ARDSArmCtrl[1].AR3slrPosition[1,1,8]													:= Arm1HookPos[1];
	ARDSArmCtrl[1].AR3slrPosition[1,2,8]													:= Arm1HookPos[2];
	ARDSArmCtrl[1].AR3slrPosition[1,3,8]													:= Arm1HookPos[3];
	ARDSArmCtrl[1].AR3slrPosition[1,4,8]													:= Arm1HookPos[4];
	ARDSArmCtrl[1].AR3slrPosition[1,5,8]													:= Arm1HookPos[5];
	ARDSArmCtrl[1].AR3slrPosition[1,6,8]													:= Arm1HookPos[6];
	ARDSArmCtrl[1].AR3slrPosition[1,7,8]													:= Arm1HookPos[7];
	ARDSArmCtrl[1].AR3slrPosition[1,8,8]													:= Arm1HookPos[8];
	ARDSArmCtrl[1].AR3slrPosition[1,9,8]													:= Arm1HookPos[9];
	ARDSArmCtrl[1].AR3slrPosition[1,10,8]													:= Arm1HookPos[10];
	ARDSArmCtrl[1].AR3slrPosition[1,11,8]													:= Arm1HookPos[11];
	ARDSArmCtrl[1].AR3slrPosition[1,12,8]													:= Arm1HookPos[12];
(*
(*ARM 2*)
	ARDSArmCtrl[2].AR3slrPosition[2,1,8];

	ARDSArmCtrl[2].AR3slrPosition[3,1,8];
	(*ARDSArmCtrl[2].AR3slrPosition[3,1,8];*)

	ARDSArmCtrl[2].AR3slrPosition[1,1,8];
	ARDSArmCtrl[2].AR3slrPosition[1,2,8];
	ARDSArmCtrl[2].AR3slrPosition[1,3,8];
	ARDSArmCtrl[2].AR3slrPosition[1,4,8];
	ARDSArmCtrl[2].AR3slrPosition[1,5,8];
	ARDSArmCtrl[2].AR3slrPosition[1,6,8];
	ARDSArmCtrl[2].AR3slrPosition[1,7,8];
	ARDSArmCtrl[2].AR3slrPosition[1,8,8];
	ARDSArmCtrl[2].AR3slrPosition[1,9,8];
	ARDSArmCtrl[2].AR3slrPosition[1,10,8];
	ARDSArmCtrl[2].AR3slrPosition[1,11,8];
	ARDSArmCtrl[2].AR3slrPosition[1,12,8];

(*On when using beckhoff HMI, Off when using Indusoft*)
(*ARM 2*)
	ARDSArmCtrl[2].AR3slrPosition[2,1,8]													:= Arm2HookPos[19];

	ARDSArmCtrl[2].AR3slrPosition[3,1,8]													:= Arm2HookPos[20];
	(*ARDSArmCtrl[2].AR3slrPosition[3,1,8];*)

	ARDSArmCtrl[2].AR3slrPosition[1,1,8]													:= Arm2HookPos[1];
	ARDSArmCtrl[2].AR3slrPosition[1,2,8]													:= Arm2HookPos[2];
	ARDSArmCtrl[2].AR3slrPosition[1,3,8]													:= Arm2HookPos[3];
	ARDSArmCtrl[2].AR3slrPosition[1,4,8]													:= Arm2HookPos[4];
	ARDSArmCtrl[2].AR3slrPosition[1,5,8]													:= Arm2HookPos[5];
	ARDSArmCtrl[2].AR3slrPosition[1,6,8]													:= Arm2HookPos[6];
	ARDSArmCtrl[2].AR3slrPosition[1,7,8]													:= Arm2HookPos[7];
	ARDSArmCtrl[2].AR3slrPosition[1,8,8]													:= Arm2HookPos[8];
	ARDSArmCtrl[2].AR3slrPosition[1,9,8]													:= Arm2HookPos[9];
	ARDSArmCtrl[2].AR3slrPosition[1,10,8]												:= Arm2HookPos[10];
	ARDSArmCtrl[2].AR3slrPosition[1,11,8]												:= Arm2HookPos[11];
	ARDSArmCtrl[2].AR3slrPosition[1,12,8]												:= Arm2HookPos[12];
*)
(*Station Unhook Postion*)
(*ARM 1*)
	ARDSArmCtrl[1].AR3slrPosition[2,1,7];

	ARDSArmCtrl[1].AR3slrPosition[3,1,7];
	(*ARDSArmCtrl[1].AR3slrPosition[3,2,7];*)

	ARDSArmCtrl[1].AR3slrPosition[1,1,7];
	ARDSArmCtrl[1].AR3slrPosition[1,2,7];
	ARDSArmCtrl[1].AR3slrPosition[1,3,7];
	ARDSArmCtrl[1].AR3slrPosition[1,4,7];
	ARDSArmCtrl[1].AR3slrPosition[1,5,7];
	ARDSArmCtrl[1].AR3slrPosition[1,6,7];
	ARDSArmCtrl[1].AR3slrPosition[1,7,7];
	ARDSArmCtrl[1].AR3slrPosition[1,8,7];
	ARDSArmCtrl[1].AR3slrPosition[1,9,7];
	ARDSArmCtrl[1].AR3slrPosition[1,10,7];
	ARDSArmCtrl[1].AR3slrPosition[1,11,7];
	ARDSArmCtrl[1].AR3slrPosition[1,12,7];

(*On when using beckhoff HMI, Off when using Indusoft*)
(*ARM 1*)
	ARDSArmCtrl[1].AR3slrPosition[2,1,7]													:= Arm1UnHookPos[19];

	ARDSArmCtrl[1].AR3slrPosition[3,1,7]													:= Arm1UnHookPos[20];
	(*ARDSArmCtrl[1].AR3slrPosition[3,2,7];*)

	ARDSArmCtrl[1].AR3slrPosition[1,1,7]													:= Arm1UnHookPos[1];
	ARDSArmCtrl[1].AR3slrPosition[1,2,7]													:= Arm1UnHookPos[2];
	ARDSArmCtrl[1].AR3slrPosition[1,3,7]													:= Arm1UnHookPos[3];
	ARDSArmCtrl[1].AR3slrPosition[1,4,7]													:= Arm1UnHookPos[4];
	ARDSArmCtrl[1].AR3slrPosition[1,5,7]													:= Arm1UnHookPos[5];
	ARDSArmCtrl[1].AR3slrPosition[1,6,7]													:= Arm1UnHookPos[6];
	ARDSArmCtrl[1].AR3slrPosition[1,7,7]													:= Arm1UnHookPos[7];
	ARDSArmCtrl[1].AR3slrPosition[1,8,7]													:= Arm1UnHookPos[8];
	ARDSArmCtrl[1].AR3slrPosition[1,9,7]													:= Arm1UnHookPos[9];
	ARDSArmCtrl[1].AR3slrPosition[1,10,7]												:= Arm1UnHookPos[10];
	ARDSArmCtrl[1].AR3slrPosition[1,11,7]												:= Arm1UnHookPos[11];
	ARDSArmCtrl[1].AR3slrPosition[1,12,7]												:= Arm1UnHookPos[12];
(*
(*ARM 2*)
	ARDSArmCtrl[2].AR3slrPosition[2,1,7];

	ARDSArmCtrl[2].AR3slrPosition[3,1,7];
	(*ARDSArmCtrl[2].AR3slrPosition[3,2,7];*)

	ARDSArmCtrl[2].AR3slrPosition[1,1,7];
	ARDSArmCtrl[2].AR3slrPosition[1,2,7];
	ARDSArmCtrl[2].AR3slrPosition[1,3,7];
	ARDSArmCtrl[2].AR3slrPosition[1,4,7];
	ARDSArmCtrl[2].AR3slrPosition[1,5,7];
	ARDSArmCtrl[2].AR3slrPosition[1,6,7];
	ARDSArmCtrl[2].AR3slrPosition[1,7,7];
	ARDSArmCtrl[2].AR3slrPosition[1,8,7];
	ARDSArmCtrl[2].AR3slrPosition[1,9,7];
	ARDSArmCtrl[2].AR3slrPosition[1,10,7];
	ARDSArmCtrl[2].AR3slrPosition[1,11,7];
	ARDSArmCtrl[2].AR3slrPosition[1,12,7];

(*On when using beckhoff HMI, Off when using Indusoft*)
(*ARM 2*)
	ARDSArmCtrl[2].AR3slrPosition[2,1,7]													:= Arm2UnHookPos[19];

	ARDSArmCtrl[2].AR3slrPosition[3,1,7]													:= Arm2UnHookPos[20];
	(*ARDSArmCtrl[2].AR3slrPosition[3,2,7];*)

	ARDSArmCtrl[2].AR3slrPosition[1,1,7]													:= Arm2UnHookPos[1];
	ARDSArmCtrl[2].AR3slrPosition[1,2,7]													:= Arm2UnHookPos[2];
	ARDSArmCtrl[2].AR3slrPosition[1,3,7]													:= Arm2UnHookPos[3];
	ARDSArmCtrl[2].AR3slrPosition[1,4,7]													:= Arm2UnHookPos[4];
	ARDSArmCtrl[2].AR3slrPosition[1,5,7]													:= Arm2UnHookPos[5];
	ARDSArmCtrl[2].AR3slrPosition[1,6,7]													:= Arm2UnHookPos[6];
	ARDSArmCtrl[2].AR3slrPosition[1,7,7]													:= Arm2UnHookPos[7];
	ARDSArmCtrl[2].AR3slrPosition[1,8,7]													:= Arm2UnHookPos[8];
	ARDSArmCtrl[2].AR3slrPosition[1,9,7]													:= Arm2UnHookPos[9];
	ARDSArmCtrl[2].AR3slrPosition[1,10,7]													:= Arm2UnHookPos[10];
	ARDSArmCtrl[2].AR3slrPosition[1,11,7]													:= Arm2UnHookPos[11];
	ARDSArmCtrl[2].AR3slrPosition[1,12,7]													:= Arm2UnHookPos[12];
*)
(*Station Up Postion*)
(*ARM 1*)
	ARDSArmCtrl[1].AR3slrPosition[2,1,1];

	ARDSArmCtrl[1].AR3slrPosition[3,1,1];
	(*ARDSArmCtrl[1].AR3slrPosition[3,2,1];*)

	ARDSArmCtrl[1].AR3slrPosition[1,1,1];
	ARDSArmCtrl[1].AR3slrPosition[1,2,1];
	ARDSArmCtrl[1].AR3slrPosition[1,3,1];
	ARDSArmCtrl[1].AR3slrPosition[1,4,1];
	ARDSArmCtrl[1].AR3slrPosition[1,5,1];
	ARDSArmCtrl[1].AR3slrPosition[1,6,1];
	ARDSArmCtrl[1].AR3slrPosition[1,7,1];
	ARDSArmCtrl[1].AR3slrPosition[1,8,1];
	ARDSArmCtrl[1].AR3slrPosition[1,9,1];
	ARDSArmCtrl[1].AR3slrPosition[1,10,1];
	ARDSArmCtrl[1].AR3slrPosition[1,11,1];
	ARDSArmCtrl[1].AR3slrPosition[1,12,1];

(*ARM 1*)
	ARDSArmCtrl[1].AR3slrPosition[2,1,1] 												:= Arm1TopPos[19];

	ARDSArmCtrl[1].AR3slrPosition[3,1,1] 												:= Arm1TopPos[20];
	(*ARDSArmCtrl[1].AR3slrPosition[3,2,1];*)

	ARDSArmCtrl[1].AR3slrPosition[1,1,1] 												:= Arm1TopPos[1];
	ARDSArmCtrl[1].AR3slrPosition[1,2,1] 												:= Arm1TopPos[2];
	ARDSArmCtrl[1].AR3slrPosition[1,3,1] 											 	:= Arm1TopPos[3];
	ARDSArmCtrl[1].AR3slrPosition[1,4,1] 												:= Arm1TopPos[4];
	ARDSArmCtrl[1].AR3slrPosition[1,5,1] 												:= Arm1TopPos[5];
	ARDSArmCtrl[1].AR3slrPosition[1,6,1] 												:= Arm1TopPos[6];
	ARDSArmCtrl[1].AR3slrPosition[1,7,1] 												:= Arm1TopPos[7];
	ARDSArmCtrl[1].AR3slrPosition[1,8,1] 												:= Arm1TopPos[8];
	ARDSArmCtrl[1].AR3slrPosition[1,9,1] 												:= Arm1TopPos[9];
	ARDSArmCtrl[1].AR3slrPosition[1,10,1] 												:= Arm1TopPos[10];
	ARDSArmCtrl[1].AR3slrPosition[1,11,1] 												:= Arm1TopPos[11];
	ARDSArmCtrl[1].AR3slrPosition[1,12,1] 												:= Arm1TopPos[12];
(*
(*ARM 2*)
	ARDSArmCtrl[2].AR3slrPosition[2,1,1];

	ARDSArmCtrl[2].AR3slrPosition[3,1,1];
	(*ARDSArmCtrl[2].AR3slrPosition[3,2,1];*)

	ARDSArmCtrl[2].AR3slrPosition[1,1,1];
	ARDSArmCtrl[2].AR3slrPosition[1,2,1];
	ARDSArmCtrl[2].AR3slrPosition[1,3,1];
	ARDSArmCtrl[2].AR3slrPosition[1,4,1];
	ARDSArmCtrl[2].AR3slrPosition[1,5,1];
	ARDSArmCtrl[2].AR3slrPosition[1,6,1];
	ARDSArmCtrl[2].AR3slrPosition[1,7,1];
	ARDSArmCtrl[2].AR3slrPosition[1,8,1];
	ARDSArmCtrl[2].AR3slrPosition[1,9,1];
	ARDSArmCtrl[2].AR3slrPosition[1,10,1];
	ARDSArmCtrl[2].AR3slrPosition[1,11,1];
	ARDSArmCtrl[2].AR3slrPosition[1,12,1];

(*ARM 2*)
	ARDSArmCtrl[2].AR3slrPosition[2,1,1] 												:= Arm2TopPos[19];

	ARDSArmCtrl[2].AR3slrPosition[3,1,1] 												:= Arm2TopPos[20];
	(*ARDSArmCtrl[2].AR3slrPosition[3,2,1];*)

	ARDSArmCtrl[2].AR3slrPosition[1,1,1] 												:= Arm2TopPos[1];
	ARDSArmCtrl[2].AR3slrPosition[1,2,1] 												:= Arm2TopPos[2];
	ARDSArmCtrl[2].AR3slrPosition[1,3,1] 											 	:= Arm2TopPos[3];
	ARDSArmCtrl[2].AR3slrPosition[1,4,1] 												:= Arm2TopPos[4];
	ARDSArmCtrl[2].AR3slrPosition[1,5,1] 												:= Arm2TopPos[5];
	ARDSArmCtrl[2].AR3slrPosition[1,6,1] 												:= Arm2TopPos[6];
	ARDSArmCtrl[2].AR3slrPosition[1,7,1] 												:= Arm2TopPos[7];
	ARDSArmCtrl[2].AR3slrPosition[1,8,1] 												:= Arm2TopPos[8];
	ARDSArmCtrl[2].AR3slrPosition[1,9,1] 												:= Arm2TopPos[9];
	ARDSArmCtrl[2].AR3slrPosition[1,10,1] 												:= Arm2TopPos[10];
	ARDSArmCtrl[2].AR3slrPosition[1,11,1] 												:= Arm2TopPos[11];
	ARDSArmCtrl[2].AR3slrPosition[1,12,1] 												:= Arm2TopPos[12];

	Arm2TopPos[6] := Arm1TopPos[6];
*)
(*Station Down Postion*)
(*ARM 1*)
	ARDSArmCtrl[1].AR3slrPosition[2,1,6];

	ARDSArmCtrl[1].AR3slrPosition[3,1,6];
	(*ARDSArmCtrl[1].AR3slrPosition[3,2,6];*)

	ARDSArmCtrl[1].AR3slrPosition[1,1,6];
	ARDSArmCtrl[1].AR3slrPosition[1,2,6];
	ARDSArmCtrl[1].AR3slrPosition[1,3,6];
	ARDSArmCtrl[1].AR3slrPosition[1,4,6];
	ARDSArmCtrl[1].AR3slrPosition[1,5,6];
	ARDSArmCtrl[1].AR3slrPosition[1,6,6];
	ARDSArmCtrl[1].AR3slrPosition[1,7,6];
	ARDSArmCtrl[1].AR3slrPosition[1,8,6];
	ARDSArmCtrl[1].AR3slrPosition[1,9,6];
	ARDSArmCtrl[1].AR3slrPosition[1,10,6];
	ARDSArmCtrl[1].AR3slrPosition[1,11,6];
	ARDSArmCtrl[1].AR3slrPosition[1,12,6];

	ARDSArmCtrl[1].AR3slrPosition[1,9,2];

(*ARM 1*)
	ARDSArmCtrl[1].AR3slrPosition[2,1,6] 												:= Arm1BottomPos[19];

	ARDSArmCtrl[1].AR3slrPosition[3,1,6] 												:= Arm1BottomPos[20];
	(*ARDSArmCtrl[1].AR3slrPosition[3,2,6];*)

	ARDSArmCtrl[1].AR3slrPosition[1,1,6] 												:= Arm1BottomPos[1];
	ARDSArmCtrl[1].AR3slrPosition[1,2,6] 												:= Arm1BottomPos[2];
	ARDSArmCtrl[1].AR3slrPosition[1,3,6] 												:= Arm1BottomPos[3];
	ARDSArmCtrl[1].AR3slrPosition[1,4,6] 												:= Arm1BottomPos[4];
	ARDSArmCtrl[1].AR3slrPosition[1,5,6] 												:= Arm1BottomPos[5];
	ARDSArmCtrl[1].AR3slrPosition[1,6,6] 												:= Arm1BottomPos[6];
	ARDSArmCtrl[1].AR3slrPosition[1,7,6] 												:= Arm1BottomPos[7];
	ARDSArmCtrl[1].AR3slrPosition[1,8,6] 												:= Arm1BottomPos[8];
	ARDSArmCtrl[1].AR3slrPosition[1,9,6]												:= Arm1BottomPos[9];
	ARDSArmCtrl[1].AR3slrPosition[1,10,6]												:= Arm1BottomPos[10];
	ARDSArmCtrl[1].AR3slrPosition[1,11,6]												:= Arm1BottomPos[11];
	ARDSArmCtrl[1].AR3slrPosition[1,12,6]												:= Arm1BottomPos[12];

	ARDSArmCtrl[1].AR3slrPosition[1,9,2]												:=Arm1MidPos[9]; (*Arm - Slow Pull Up Position*)
(*
(*ARM 2*)
	ARDSArmCtrl[2].AR3slrPosition[2,1,6];

	ARDSArmCtrl[2].AR3slrPosition[3,1,6];
	(*ARDSArmCtrl[2].AR3slrPosition[3,2,6];*)

	ARDSArmCtrl[2].AR3slrPosition[1,1,6];
	ARDSArmCtrl[2].AR3slrPosition[1,2,6];
	ARDSArmCtrl[2].AR3slrPosition[1,3,6];
	ARDSArmCtrl[2].AR3slrPosition[1,4,6];
	ARDSArmCtrl[2].AR3slrPosition[1,5,6];
	ARDSArmCtrl[2].AR3slrPosition[1,6,6];
	ARDSArmCtrl[2].AR3slrPosition[1,7,6];
	ARDSArmCtrl[2].AR3slrPosition[1,8,6];
	ARDSArmCtrl[2].AR3slrPosition[1,9,6];
	ARDSArmCtrl[2].AR3slrPosition[1,10,6];
	ARDSArmCtrl[2].AR3slrPosition[1,11,6];
	ARDSArmCtrl[2].AR3slrPosition[1,12,6];

	ARDSArmCtrl[2].AR3slrPosition[1,8,2]; (*Arm - Slow Pull Up Position*)

(*ARM 2*)
	ARDSArmCtrl[2].AR3slrPosition[2,1,6] 												:= Arm2BottomPos[19];

	ARDSArmCtrl[2].AR3slrPosition[3,1,6] 												:= Arm2BottomPos[20];
	(*ARDSArmCtrl[2].AR3slrPosition[3,2,6];*)

	ARDSArmCtrl[2].AR3slrPosition[1,1,6] 												:= Arm2BottomPos[1];
	ARDSArmCtrl[2].AR3slrPosition[1,2,6] 												:= Arm2BottomPos[2];
	ARDSArmCtrl[2].AR3slrPosition[1,3,6] 												:= Arm2BottomPos[3];
	ARDSArmCtrl[2].AR3slrPosition[1,4,6] 												:= Arm2BottomPos[4];
	ARDSArmCtrl[2].AR3slrPosition[1,5,6] 												:= Arm2BottomPos[5];
	ARDSArmCtrl[2].AR3slrPosition[1,6,6] 												:= Arm2BottomPos[6];
	ARDSArmCtrl[2].AR3slrPosition[1,7,6] 												:= Arm2BottomPos[7];
	ARDSArmCtrl[2].AR3slrPosition[1,8,6] 												:= Arm2BottomPos[8];
	ARDSArmCtrl[2].AR3slrPosition[1,9,6]												:= Arm2BottomPos[9];
	ARDSArmCtrl[2].AR3slrPosition[1,10,6]												:= Arm2BottomPos[10];
	ARDSArmCtrl[2].AR3slrPosition[1,11,6]												:= Arm2BottomPos[11];
	ARDSArmCtrl[2].AR3slrPosition[1,12,6]												:= Arm2BottomPos[12];

	ARDSArmCtrl[2].AR3slrPosition[1,8,2];

	Arm2BottomPos[6] := Arm1BottomPos[6];
*)

(*Loading & Unloading Station & Station Centre-Hook Position - for fbV2_FBPArmHorzZoneConfirm*)

(*ARM 1*)
	ARlrLdHorzCentrePoint[1] 															:= ARDSArmCtrl[1].AR3slrPosition[2,1,8];

	ARlrUldHorzCentrePoint[1] 															:= ARDSArmCtrl[1].AR3slrPosition[3,1,8];
	(*ARlrUldHorzCentrePoint[2] 														:= ARDSArmCtrl[1].AR3slrPosition[3,2,8];*)

	ARlrStnHorzCentrePoint[1] 															:= ARDSArmCtrl[1].AR3slrPosition[1,1,8];
	ARlrStnHorzCentrePoint[2] 															:= ARDSArmCtrl[1].AR3slrPosition[1,2,8];
	ARlrStnHorzCentrePoint[3] 															:= ARDSArmCtrl[1].AR3slrPosition[1,3,8];
	ARlrStnHorzCentrePoint[4] 															:= ARDSArmCtrl[1].AR3slrPosition[1,4,8];
	ARlrStnHorzCentrePoint[5] 															:= ARDSArmCtrl[1].AR3slrPosition[1,5,8];
	ARlrStnHorzCentrePoint[6] 															:= ARDSArmCtrl[1].AR3slrPosition[1,6,8];
	ARlrStnHorzCentrePoint[7] 															:= ARDSArmCtrl[1].AR3slrPosition[1,7,8];
	ARlrStnHorzCentrePoint[8] 															:= ARDSArmCtrl[1].AR3slrPosition[1,8,8];
	ARlrStnHorzCentrePoint[9] 															:= ARDSArmCtrl[1].AR3slrPosition[1,9,8];
	ARlrStnHorzCentrePoint[10] 															:= ARDSArmCtrl[1].AR3slrPosition[1,10,8];
	ARlrStnHorzCentrePoint[11] 															:= ARDSArmCtrl[1].AR3slrPosition[1,11,8];
	ARlrStnHorzCentrePoint[12] 															:= ARDSArmCtrl[1].AR3slrPosition[1,12,8];

(*ARM 2*)
	ARlrArm2LdHorzCentrePoint[1] 														:= ARDSArmCtrl[2].AR3slrPosition[2,1,8];

	ARlrArm2UldHorzCentrePoint[1] 														:= ARDSArmCtrl[2].AR3slrPosition[3,1,8];
	(*ARlrArm2UldHorzCentrePoint[2] 													:= ARDSArmCtrl[2].AR3slrPosition[3,2,8];*)

	ARlrArm2StnHorzCentrePoint[1] 														:= ARDSArmCtrl[2].AR3slrPosition[1,1,8];
	ARlrArm2StnHorzCentrePoint[2] 														:= ARDSArmCtrl[2].AR3slrPosition[1,2,8];
	ARlrArm2StnHorzCentrePoint[3] 														:= ARDSArmCtrl[2].AR3slrPosition[1,3,8];
	ARlrArm2StnHorzCentrePoint[4] 														:= ARDSArmCtrl[2].AR3slrPosition[1,4,8];
	ARlrArm2StnHorzCentrePoint[5] 														:= ARDSArmCtrl[2].AR3slrPosition[1,5,8];
	ARlrArm2StnHorzCentrePoint[6] 														:= ARDSArmCtrl[2].AR3slrPosition[1,6,8];
	ARlrArm2StnHorzCentrePoint[7] 														:= ARDSArmCtrl[2].AR3slrPosition[1,7,8];
	ARlrArm2StnHorzCentrePoint[8] 														:= ARDSArmCtrl[2].AR3slrPosition[1,8,8];
	ARlrArm2StnHorzCentrePoint[9] 														:= ARDSArmCtrl[2].AR3slrPosition[1,9,8];
	ARlrArm2StnHorzCentrePoint[10] 														:= ARDSArmCtrl[2].AR3slrPosition[1,10,8];
	ARlrArm2StnHorzCentrePoint[11] 														:= ARDSArmCtrl[2].AR3slrPosition[1,11,8];
	ARlrArm2StnHorzCentrePoint[12]														:= ARDSArmCtrl[2].AR3slrPosition[1,12,8];


(*xxxxxxxxxxxxxxxxxxxxxxxxxxxxxxxxxx Inverter with Encoder Ctrl xxxxxxxxxxxxxxxxxxxxxxxxxxxxxxxxxx*)
(*Inverter Encoder &  HzToRaw Ratio Variable Ctrl*)
	ARlrVertRatioPulseToMM[1]														(*:= 40.01775*);
	ARlrHorzRatioPulseToMM[1]														(*:= 40.64147*);

	ARiVertCounterValueResetTime_Sec[1];
	ARiHorzCounterValueResetTime_Sec[1];

	ARrVertGen_In_HzToRawRatio[1]													:= 327.67;
	ARrHorzGen_In_HzToRawRatio[1]													:= 327.67;

(*Arm Positioning Variable Ctrl*)
	ARlrArmVertFix_PosCfmTolerance[1]													(*:= 2*);
	ARlrArmVertFix_2ndSpdRange[1]													(*:= 100*);

	ARlrArmHorzFix_PosCfmTolerance[1]												(*:= 3*);
	ARlrArmHorzFix_2ndSpdRange[1]													(*:= 115*);

(*Arm Pos Variable Ctrl*)
	ARrVertPos_In_TargetSpdHz[1]														(*:= 50*);
	ARrVertPos_In_2ndSpdHz[1]														(*:= 5*);

	ARrHorzPos_In_TargetSpdHz[1]														(*:= 10*);
	ARrHorzPos_In_2ndSpdHz[1]														(*:= 3*);


(*xxxxxxxxxxxxxxxxxxxxxxxxxxxxxxxxxx Servo Ctrl xxxxxxxxxxxxxxxxxxxxxxxxxxxxxxxxxx*)
(*Arm Home Variable Ctrl*)
(*ARM 1*) (*servo drive- mm/sec*)
	ARrArmVertHome1stPercent[1]														:= 50;
	ARrArmVertHome2ndPercent[1]														:= 5;
	ARrVertHomeDccDelayTimeSec[1]													:= 0.1;

	ARrArmVertHome1stPercentAcc[1]													:= 1500;
	ARrArmVertHome1stPercentDcc[1]													:= 1500;
	ARrArmVertHome2ndPercentAcc[1]													:= 1500;
	ARrArmVertHome2ndPercentDcc[1]													:= 1500;

	ARrArmHorzHome1stPercent[1]														:= 70;
	ARrArmHorzHome2ndPercent[1]														:= 5;
	ARrHorzHomeDccDelayTimeSec[1]													:= 0.1;

	ARrArmHorzHome1stPercentAcc[1]													:= 1500;
	ARrArmHorzHome1stPercentDcc[1]													:= 1500;
	ARrArmHorzHome2ndPercentAcc[1]													:= 1500;
	ARrArmHorzHome2ndPercentDcc[1]													:= 1500;

(*ARM 2*)
	ARrArmVertHome1stPercent[2]														:= 50;
	ARrArmVertHome2ndPercent[2]														:= 5;
	ARrVertHomeDccDelayTimeSec[2]													:= 0.1;

	ARrArmVertHome1stPercentAcc[2]													:= 1500;
	ARrArmVertHome1stPercentDcc[2]													:= 1500;
	ARrArmVertHome2ndPercentAcc[2]													:= 1500;
	ARrArmVertHome2ndPercentDcc[2]													:= 1500;

	ARrArmHorzHome1stPercent[2]														:= 70;
	ARrArmHorzHome2ndPercent[2]														:= 5;
	ARrHorzHomeDccDelayTimeSec[2]													:= 0.1;

	ARrArmHorzHome1stPercentAcc[2]													:= 1500;
	ARrArmHorzHome1stPercentDcc[2]													:= 1500;
	ARrArmHorzHome2ndPercentAcc[2]													:= 1500;
	ARrArmHorzHome2ndPercentDcc[2]													:= 1500;

(*Slow Pull*)
	DSHomingSetting.lrArmLifterHomeVelo												:= 5;
	DSHomingSetting.lrArmLifterHomeAcc												:= 200;
	DSHomingSetting.lrArmLifterHomeDcc												:= 200;

	DSHomingSetting.lrArmLifter2HomeVelo											:= 3;
	DSHomingSetting.lrArmLifter2HomeAcc												:= 200;
	DSHomingSetting.lrArmLifter2HomeDcc												:= 200;


(*Arm Jog Variable Ctrl*)
(*ARM 1*) (*servo drive - mm/sec*)
	ARrArmVertJogPercent[1]; 		ARrArmHorzJogPercent[1];
	ARrArmVertJogAcc[1]; 			ARrArmHorzJogAcc[1];
	ARrArmVertJogDcc[1]; 			ARrArmHorzJogDcc[1];

(*ARM 2*)
	ARrArmVertJogPercent[2]; 		ARrArmHorzJogPercent[2];
	ARrArmVertJogAcc[2]; 			ARrArmHorzJogAcc[2];
	ARrArmVertJogDcc[2]; 			ARrArmHorzJogDcc[2];

(*Slow Pull*)
	ARlrArmSlowPullJogVelo[1];
	ARlrArmSlowPullJogAcc[1];
	ARlrArmSlowPullJogDcc[1];


(*Arm Pos Variable Ctrl*)
(*ARM 1*)
	ARlrVertPos_In_HighSpeed[1]; 		ARlrHorzPos_In_HighSpeed[1];
	ARlrVertPos_In_Acc[1]; 			ARlrHorzPos_In_Acc[1];
	ARlrVertPos_In_Dcc[1]; 			ARlrHorzPos_In_Dcc[1];

(*ARM 2*)
	ARlrVertPos_In_HighSpeed[2]; 		ARlrHorzPos_In_HighSpeed[2];
	ARlrVertPos_In_Acc[2]; 			ARlrHorzPos_In_Acc[2];
	ARlrVertPos_In_Dcc[2]; 			ARlrHorzPos_In_Dcc[2];

(*Slow Pull*)
	DS_ArmLifterPosition.lrSlowPullDownVelo;
	DS_ArmLifterPosition.lrSlowPullDownAcc;
	DS_ArmLifterPosition.lrSlowPullDownDcc;

	DS_ArmLifterPosition.lrSlowPullDown2ndVelo											:= 3;
	DS_ArmLifterPosition.lrSlowPullDown2ndAcc											:= 200;
	DS_ArmLifterPosition.lrSlowPullDown2ndDcc											:= 200;

	DS_ArmLifterPosition.lrSlowPullUpVelo;
	DS_ArmLifterPosition.lrSlowPullUpAcc;
	DS_ArmLifterPosition.lrSlowPullUpDcc;

	DS_ArmLifterPosition.lrSlowPullUp2ndVelo											:= 3;
	DS_ArmLifterPosition.lrSlowPullUp2ndAcc												:= 200;
	DS_ArmLifterPosition.lrSlowPullUp2ndDcc												:= 200;


(*Station Tolerance Time Variable Ctrl - Overtime to determine BAD Basket*)

(*ARM 1*) (*normally set with 60sec*)
	ARiStnToleranceTimeSV[1];
	ARiStnToleranceTimeSV[2];
	ARiStnToleranceTimeSV[3];
	ARiStnToleranceTimeSV[4];
	ARiStnToleranceTimeSV[5];
	ARiStnToleranceTimeSV[6];
	ARiStnToleranceTimeSV[7];
	ARiStnToleranceTimeSV[8];
	ARiStnToleranceTimeSV[9];
	ARiStnToleranceTimeSV[10];
	ARiStnToleranceTimeSV[11];
	ARiStnToleranceTimeSV[12];

(*ARM 1 alarm - arm overrtime alarm*) (*normally set 30sec*)
	ARiArmToleranceTimeSV[1];

(*ARM 2*)
	ARiArmToleranceTimeSV[2];


(*Station Dipping Time Variable Ctrl - AutoMode Pnp Dipping Time*)
	ARiStnDippingTimeSV[1];
	ARiStnDippingTimeSV[2];
	ARiStnDippingTimeSV[3];
	ARiStnDippingTimeSV[4];
	ARiStnDippingTimeSV[5];
	ARiStnDippingTimeSV[6];
	ARiStnDippingTimeSV[7];
	ARiStnDippingTimeSV[8];
	ARiStnDippingTimeSV[9];
	ARiStnDippingTimeSV[10];
	ARiStnDippingTimeSV[11];
	ARiStnDippingTimeSV[12];


(*Station Top Up Delay Off Time Variable Ctrl*)
	ARiStnTopUpDelayOffTimeSV[1];
	ARiStnTopUpDelayOffTimeSV[2];
	ARiStnTopUpDelayOffTimeSV[3];
	ARiStnTopUpDelayOffTimeSV[4];
	ARiStnTopUpDelayOffTimeSV[5];
	ARiStnTopUpDelayOffTimeSV[6];
	ARiStnTopUpDelayOffTimeSV[7];
	ARiStnTopUpDelayOffTimeSV[8];
	ARiStnTopUpDelayOffTimeSV[9];
	ARiStnTopUpDelayOffTimeSV[10];
	ARiStnTopUpDelayOffTimeSV[11];
	ARiStnTopUpDelayOffTimeSV[12];

	ARiStnSubTankTopUpDelayOffTimeSV[1];
	ARiStnSubTankTopUpDelayOffTimeSV[2];
	ARiStnSubTankTopUpDelayOffTimeSV[3];
	ARiStnSubTankTopUpDelayOffTimeSV[4];
	ARiStnSubTankTopUpDelayOffTimeSV[5];
	ARiStnSubTankTopUpDelayOffTimeSV[6];
	ARiStnSubTankTopUpDelayOffTimeSV[7];
	ARiStnSubTankTopUpDelayOffTimeSV[8];
	ARiStnSubTankTopUpDelayOffTimeSV[9];
	ARiStnSubTankTopUpDelayOffTimeSV[10];
	ARiStnSubTankTopUpDelayOffTimeSV[11];
	ARiStnSubTankTopUpDelayOffTimeSV[12];


(*Arm Mishook Sensor Detect Zone Variable Ctrl*)
(*ARM 1*) (*normally set 200 - non-detection area., from bottom *)
	ARlrArmDetectZoneRange[1];
	ARlrArmDetectZoneRange[2];
	ARlrArmDetectZoneRange[3];
	ARlrArmDetectZoneRange[4];
	ARlrArmDetectZoneRange[5];
	ARlrArmDetectZoneRange[6];
	ARlrArmDetectZoneRange[7];
	ARlrArmDetectZoneRange[8];
	ARlrArmDetectZoneRange[9];
	ARlrArmDetectZoneRange[10];
	ARlrArmDetectZoneRange[11];
	ARlrArmDetectZoneRange[12];

(*if set more than the bottom position value, will not monitor this misshook function*)
	ARiArmDeactDetectZoneRange[1];

(*	ARlrArmStnDetectZoneRange[2,10] := 300;*)

(*ARM 2*)
	ARiArmDeactDetectZoneRange[2];


(*Station Call Arm Time Variable Ctrl*)

	tAllStnArmTake;


(*Unloading Buzzer Time Variable Ctrl*)

	diUnloadingTimer;


(*Alternate Station Variable Ctrl*)

	ARbAlternateStnEn [1] ;
	ARbAlternateStnEn [2] ;

